//PRZYPISANIE BŁĘDÓW STACJI DO TABLICY 
aStationsErrors[1]															:=GeneralAlarms;											
aStationsErrors[2]															:=FormTransporterDispencerError;					//E_ConveyorState			// Transporter wjazdowy pod dozowniki
aStationsErrors[3]															:=FormTransporterScrewerError;						//E_ConveyorState			// Transporter wyjazdowy spod dozowników
aStationsErrors[4]															:=DispencersDragLeftError;							//E_DragStationState		// Przeciąganie formatek pod dozownikami
aStationsErrors[5]															:=DispencersCatch1Error;							//E_CatchStationState		// Chwytak butelek dozownika nr.1
aStationsErrors[6]															:=DispencersCatch2Error;							//E_CatchStationState		// Chwytak butelek dozownika nr.2
aStationsErrors[7]															:=DispencersCatch3Error;							//E_CatchStationState		// Chwytak butelek dozownika nr.3
aStationsErrors[8]															:=DispencersCatch4Error;							//E_CatchStationState		// Chwytak butelek dozownika nr.4				
aStationsErrors[9]															:=Dispencer1Error;									//E_DispencerState			// Dozownik 1
aStationsErrors[10]															:=Dispencer2Error;									//E_DispencerState			// Dozownik 2
aStationsErrors[11]															:=Dispencer3Error;									//E_DispencerState			// Dozownik 3							
aStationsErrors[12]															:=Dispencer4Error;									//E_DispencerState			// Dozownik 4
aStationsErrors[13]															:=TankHeatingError;									//E_MassHeatingState		// Grzanie masy
aStationsErrors[14]															:=WeightLiftError;									//E_WeightLiftState			// Podnoszenie wideł i szalek
aStationsErrors[15]															:=Weight1Error;										//E_WeightState				// Waga 1
aStationsErrors[16]															:=Weight2Error;										//E_WeightState				// Waga 2
aStationsErrors[17]															:=Weight3Error;										//E_WeightState				// Waga 3
aStationsErrors[18]															:=Weight4Error;										//E_WeightState				// Waga 4
aStationsErrors[19]															:=Dispencer1CorrectionError;						//E_WeightCorrectionState	//Korketa wagi 
aStationsErrors[20]															:=Dispencer2CorrectionError;						//E_WeightCorrectionState	//Korketa wagi 
aStationsErrors[21]															:=Dispencer3CorrectionError;						//E_WeightCorrectionState	//Korketa wagi 
aStationsErrors[22]															:=Dispencer4CorrectionError;						//E_WeightCorrectionState	//Korketa wagi 
aStationsErrors[23]															:=CapPuttedCheckError;								//E_CheckerState			// Sprawdzenie nałożenia nasadki
aStationsErrors[24]															:=GripperScrewerCatch1Error;						//E_CatchStationState 		// Łapanie butelek pod zakręcarkami 1
aStationsErrors[25]															:=GripperScrewerCatch2Error;						//E_CatchStationState 		// Łapanie butelek pod zakręcarkami	2
aStationsErrors[26]															:=GripperScrewer1Error;								//E_GriperScrewer			// Zakręcarka szczękowa 1
aStationsErrors[27]															:=GripperScrewer2Error;											
aStationsErrors[28]															:=BottleDragError;									//E_DragStationState		// Przeciąganie butelek pod zakręcarkami
aStationsErrors[29]															:=CapCorrectCheckError;								// E_CheckerState			// Sprawdzenie poprawności zakręcenia	
aStationsErrors[30]															:=BottleTransferError;								//E_BottleTransferState		// Robot
aStationsErrors[31]															:=GateRobotError;									// 							// Szlaban pod roobtem
aStationsErrors[32]															:=BadBottleConveyorError;							//E_ConvoyerState			// Stan transportera odrzuconych
aStationsErrors[33]															:=LabelMachineError;								// 							// Stan etykieciarki
aStationsErrors[34]															:=TanksError;										// 							// Stan zbiorników
aStationsErrors[35]															:=ExitTurnTableError;								//							// Stan stołu oboortowego wujscia z etykieciakri
aStationsErrors[36]															:=FormTransporterBeforeScrewerError;				//							// Spowalniacz formatek
aStationsErrors[37]															:=CapFeederError;									// Podajnik nasadek
aStationsErrors[38]															:=Weight5Error;										//E_WeightState				// Waga 5 	(** dodane 07.04.2022**)
aStationsErrors[39]															:=Weight6Error;										//E_WeightState				// Waga 6 	(** dodane 07.04.2022**)
aStationsErrors[40]															:=BottleFeederError;								// E_BottleFeederState     (** dodane 13.04.2022**)
aStationsErrors[41]															:=DispencersDragRightError;							//							// Przeciąganie formatek pod dozownikami prawa storna
aStationsErrors[42]															:=BarrierBetweenDispencers;							// 							//	Szlaban pod dozownikami od dwufazy
aStationsErrors[43]															:=BarrierBetweenWeights;
aStationsErrors[44]															:=BottleFeederTurnTableError;						//							//	Szlaban pomiedzy wagami od dwufazy
aStationsErrors[45]															:=BottleFeederFormGateError;
aStationsErrors[46]															:=SensorAcetoneError;
aStationsErrors[47]															:=SensorAirFlowError;
aStationsErrors[48]															:=LidFeederFormPositioningError;

aStationsErrors[49].bReset;
aStationsErrors[49].bError													:= stBottleSorterRead.eError.bError;
aStationsErrors[49].nErrorCode												:= stBottleSorterRead.eError.nErrorCode;
aStationsErrors[49].sErrorString											:= stBottleSorterRead.eError.sErrorString;
aStationsErrors[49].sErrorString2											:= stBottleSorterRead.eError.sErrorString2;
aStationsErrors[49].udiStationID											:= stBottleSorterRead.eError.udiStationID;
aStationsErrors[49].sStationName											:= Concat('Sorter butelek | ',stBottleSorterRead.eError.sStationName);

aStationsErrors[50].bReset;
aStationsErrors[50].bError													:= stCapSorterRead.eError.bError;
aStationsErrors[50].nErrorCode												:= stCapSorterRead.eError.nErrorCode;
aStationsErrors[50].sErrorString											:= stCapSorterRead.eError.sErrorString;
aStationsErrors[50].sErrorString2											:= stCapSorterRead.eError.sErrorString2;
aStationsErrors[50].udiStationID											:= stCapSorterRead.eError.udiStationID;
aStationsErrors[50].sStationName											:= Concat('Sorter nasadek | ',stCapSorterRead.eError.sStationName);

aStationsErrors[51]															:=CapSorterDragError;									
aStationsErrors[52]															:=BottlePusherError;									

aStationsErrors[53]															:=BarrierLidFeeder;	
aStationsErrors[54]															:=LidFeederError;		
aStationsErrors[55]															:=LidFeeder2Error;		
aStationsErrors[56]															:=LidFeederDragError;
aStationsErrors[57]															:=CapCorrectCheckCameraError;
aStationsErrors[58]															:=LidSealerError;		
aStationsErrors[59]															:=LidSealer2Error;		
aStationsErrors[60]															:=LidSealerDragError;

aStationsErrors[61]															:=PucksInserterError;		
aStationsErrors[62]															:=//PucksInserterTurnTableError;
aStationsErrors[63]															:=PucksInserterFormGateError;

aStationsErrors[64]															:=ROPPSlowerError;	
aStationsErrors[65]															:=ROPPFeederError;	
aStationsErrors[66]															:=ROPPDragError;	
aStationsErrors[67]															:=ROPPCappingError;
aStationsErrors[68]															:=FormTransporterROPPError;
aStationsErrors[69]															:=FormTransporterSlowerError;
aStationsErrors[70]															:=ExitConveyorError;
aStationsErrors[71]															:=SensorAcetoneError;
aStationsErrors[72]															:=SensorAirFlowError;
aStationsErrors[73]															:=ExhaustFanError;
aStationsErrors[79]															:= PucksInserterPushTableError_m1;
aStationsErrors[80]															:= PucksInserterPushTableError_m2;
aStationsErrors[81]															:= PucksInserterPushTableError_m3;
aStationsErrors[82];
aStationsErrors[83]															:= FormTransporterAfterScrewerError;
//Przegląd czy jakaś stacja jest w stanie błędu
aStationsErrors[84]															:= BottleTransferAfterDragError;
aStationsErrors[85] 														:= WickFeederError;
aStationsErrors[86]															:= WickFeederDragError;
aStationsErrors[87]															:= FormTransporterAfterCapSorterError;
aStationsErrors[88]															:= FormTransporterAfterBottleTransferError;
FOR i:=1 TO STATION_COUNT DO
	//Jeśli w stanie błędu
	
	IF aStationsErrors[i].bError THEN
		
		tonResetOff(IN:=bResetError,PT:=T#2S);
		
		IF tonResetOff.Q THEN
			aStationsErrors[i].bReset										:=FALSE;
			bResetError														:=FALSE;
		END_IF
		
		IF VIS.bResetErrorVisuCmd THEN
			aStationsErrors[i].bReset										:=TRUE;
			VIS.bResetErrorVisuCmd											:=FALSE;
		END_IF
		
		VIS.bErrorOccure													:=aStationsErrors[i].bError;
		bResetError															:=aStationsErrors[i].bReset;
		VIS.udiStationInError												:=aStationsErrors[i].udiStationID;
		VIS.sStationInError													:=aStationsErrors[i].sStationName;
		VIS.udiStationErrorCode												:=aStationsErrors[i].nErrorCode;
		VIS.sStationErrorDescription										:=aStationsErrors[i].sErrorString;
		VIS.sStationErrorDescription2										:=aStationsErrors[i].sErrorString2;
		EXIT;
		
	ELSE
		tonResetOff(IN:=bResetError,PT:=T#2S);
		//Jesli nie
		aStationsErrors[i].bError											:=FALSE;
		aStationsErrors[i].bReset											:=FALSE;
		aStationsErrors[i].sStationName										:='';
		aStationsErrors[i].nErrorCode										:=0;
		aStationsErrors[i].sErrorString										:='';
		aStationsErrors[i].sErrorString2									:='';
		VIS.bErrorOccure													:=FALSE;
	END_IF
	
	IF i>=60 THEN
		bResetError															:=FALSE;
	END_IF
	
END_FOR

// Zachowanie linii po wystapieniu błędu
IF VIS.bErrorOccure THEN
    VIS.bCycleStart 														:= FALSE; //DO WIZARDA
ELSE
    VIS.bErrorOccure              											:= FALSE;
    bResetError                  											:= FALSE;
    VIS.sStationInError           											:= '';
	VIS.udiStationInError													:=	0;
    VIS.udiStationErrorCode         										:= 0;
    VIS.sStationErrorDescription  											:= '';
    VIS.sStationErrorDescription2 											:= '';
    VIS.bResetErrorVisuCmd        											:= FALSE;
END_IF

// 
GeneralAlarms						:=aStationsErrors[1];										
FormTransporterDispencerError		:=aStationsErrors[2];					//E_ConveyorState			// Transporter wjazdowy pod dozowniki
FormTransporterScrewerError			:=aStationsErrors[3];					//E_ConveyorState			// Transporter wyjazdowy spod dozowników
DispencersDragLeftError				:=aStationsErrors[4];					//E_DragStationState		// Przeciąganie formatek pod dozownikami
DispencersCatch1Error				:=aStationsErrors[5];					//E_CatchStationState		// Chwytak butelek dozownika nr.1
DispencersCatch2Error				:=aStationsErrors[6];					//E_CatchStationState		// Chwytak butelek dozownika nr.2
DispencersCatch3Error				:=aStationsErrors[7];					//E_CatchStationState		// Chwytak butelek dozownika nr.3
DispencersCatch4Error				:=aStationsErrors[8];					//E_CatchStationState		// Chwytak butelek dozownika nr.4				
Dispencer1Error						:=aStationsErrors[9];					//E_DispencerState			// Dozownik 1
Dispencer2Error						:=aStationsErrors[10];					//E_DispencerState			// Dozownik 2
Dispencer3Error						:=aStationsErrors[11];					//E_DispencerState			// Dozownik 3							
Dispencer4Error						:=aStationsErrors[12];					//E_DispencerState			// Dozownik 4
TankHeatingError					:=aStationsErrors[13];					//E_MassHeatingState		// Grzanie masy
WeightLiftError						:=aStationsErrors[14];					//E_WeightLiftState			// Podnoszenie wideł i szalek
Weight1Error						:=aStationsErrors[15];					//E_WeightState				// Waga 1
Weight2Error						:=aStationsErrors[16];					//E_WeightState				// Waga 2
Weight3Error						:=aStationsErrors[17];					//E_WeightState				// Waga 3
Weight4Error						:=aStationsErrors[18];					//E_WeightState				// Waga 4
Dispencer1CorrectionError			:=aStationsErrors[19];				
Dispencer2CorrectionError			:=aStationsErrors[20];	
Dispencer3CorrectionError			:=aStationsErrors[21];	
Dispencer4CorrectionError			:=aStationsErrors[22];		
CapPuttedCheckError					:=aStationsErrors[23];					//E_CheckerState			// Sprawdzenie nałożenia nasadki
GripperScrewerCatch1Error			:=aStationsErrors[24];					//E_CatchStationState 		// Łapanie butelek pod zakręcarkami 1
GripperScrewerCatch2Error			:=aStationsErrors[25];					//E_CatchStationState 		// Łapanie butelek pod zakręcarkami	2
GripperScrewer1Error				:=aStationsErrors[26];					//E_GriperScrewer			// Zakręcarka szczękowa 1
GripperScrewer2Error			  	:=aStationsErrors[27];					//E_GriperScrewer			// Byyła Zakręcarka szczękowa 2;							
BottleDragError						:=aStationsErrors[28];					//E_DragStationState		// Przeciąganie butelek pod zakręcarkami
CapCorrectCheckError				:=aStationsErrors[29];					//E_CheckerState			// Sprawdzenie poprawności zakręcenia	
BottleTransferError					:=aStationsErrors[30];					// Robot
GateRobotError						:=aStationsErrors[31];			
BadBottleConveyorError				:=aStationsErrors[32];			
LabelMachineError					:=aStationsErrors[33];	
TanksError							:=aStationsErrors[34];	
ExitTurnTableError					:=aStationsErrors[35];	
FormTransporterBeforeScrewerError	:=aStationsErrors[36];	
CapFeederError						:=aStationsErrors[37];					// Podajnik nakrętek
Weight5Error						:=aStationsErrors[38];  				(** dodane 07.04.2022**)
Weight6Error						:=aStationsErrors[39];					(** dodane 07.04.2022**)
BottleFeederError					:=aStationsErrors[40];					(** dodane 13.04.2022**)
DispencersDragRightError			:=aStationsErrors[41];	
BarrierBetweenDispencers			:=aStationsErrors[42];
BarrierBetweenWeights				:=aStationsErrors[43];
BottleFeederTurnTableError			:=aStationsErrors[44];
BottleFeederFormGateError				:=aStationsErrors[45];
SensorAcetoneError 					:=aStationsErrors[46];
SensorAirFlowError 					:=aStationsErrors[47];
LidFeederFormPositioningError		:=aStationsErrors[48];	
stBottleSorterWrite.eError.bReset   :=aStationsErrors[49].bReset;						
stCapSorterWrite.eError.bReset   	:=aStationsErrors[50].bReset;	
CapSorterDragError					:=aStationsErrors[51];		
BottlePusherError					:=aStationsErrors[52];		
BarrierLidFeeder					:=aStationsErrors[53];												
LidFeederError						:=aStationsErrors[54];												
LidFeeder2Error						:=aStationsErrors[55];												
LidFeederDragError					:=aStationsErrors[56];											
CapCorrectCheckCameraError			:=aStationsErrors[57];											
LidSealerError						:=aStationsErrors[58];												
LidSealer2Error						:=aStationsErrors[59];												
LidSealerDragError					:=aStationsErrors[60];											

PucksInserterError					:=aStationsErrors[61];
//PucksInserterTurnTableError			:=aStationsErrors[62];
PucksInserterFormGateError			:=aStationsErrors[63];
ROPPSlowerError 					:=aStationsErrors[64];			
ROPPFeederError 					:=aStationsErrors[65];
ROPPDragError 						:=aStationsErrors[66];
ROPPCappingError 					:=aStationsErrors[67];
FormTransporterROPPError			:=aStationsErrors[68];
FormTransporterSlowerError			:=aStationsErrors[69];
ExitConveyorError					:=aStationsErrors[70];
SensorAcetoneError					:=aStationsErrors[71];
SensorAirFlowError					:=aStationsErrors[72];
ExhaustFanError						:=aStationsErrors[73];
PucksInserterPushTableError_m1		:=aStationsErrors[79];								
PucksInserterPushTableError_m2		:=aStationsErrors[80];								
PucksInserterPushTableError_m3		:=aStationsErrors[81];
									aStationsErrors[82];
FormTransporterAfterScrewerError	:=aStationsErrors[83];
BottleTransferAfterDragError		:=aStationsErrors[84];
WickFeederError						:=aStationsErrors[85];
WickFeederDragError					:=aStationsErrors[86];
FormTransporterAfterCapSorterError	:= aStationsErrors[87];	
FormTransporterAfterBottleTransferError := aStationsErrors[88];
//Przepisywanie ostatnich błędów
IF rtMachineStateAborting.Q THEN
    nCountSaveLastError := nCountSaveLastError + 1;
    aLastStationsErrors := aStationsErrors;
END_IF
IF P00_PackML.fbPMLAuto.ePMLState = Tc3_PackML.E_PMLState.ePMLState_EXECUTE THEN
	aLastStationsErrors := aStationsErrors;
END_IF
aStationsErrors[30].breset;

ACTION aActiveWarnings:
//	AwsActiveWarningDescription								:ARRAY [0..63] OF STRING;	//  Aktywne ostrzeżenia
//	iActiveWarning											:INT;	// Ilość aktywnych ostrzeżeń		


AbActiveWarningDescription[0]	:=	VIS.uliWarningOccure.0;
AbActiveWarningDescription[1]	:=	VIS.uliWarningOccure.1;
AbActiveWarningDescription[2]	:=	VIS.uliWarningOccure.2;
AbActiveWarningDescription[3]	:=	VIS.uliWarningOccure.3;
AbActiveWarningDescription[4]	:=	VIS.uliWarningOccure.4;
AbActiveWarningDescription[5]	:=	VIS.uliWarningOccure.5;
AbActiveWarningDescription[6]	:=	VIS.uliWarningOccure.6;
AbActiveWarningDescription[7]	:=	VIS.uliWarningOccure.7;
AbActiveWarningDescription[8]	:=	VIS.uliWarningOccure.8;
AbActiveWarningDescription[9]	:=	VIS.uliWarningOccure.9;
AbActiveWarningDescription[10]	:=	VIS.uliWarningOccure.10;
AbActiveWarningDescription[11]	:=	VIS.uliWarningOccure.11;
AbActiveWarningDescription[12]	:=	VIS.uliWarningOccure.12;
AbActiveWarningDescription[13]	:=	VIS.uliWarningOccure.13;
AbActiveWarningDescription[14]	:=	VIS.uliWarningOccure.14;
AbActiveWarningDescription[15]	:=	VIS.uliWarningOccure.15;
AbActiveWarningDescription[16]	:=	VIS.uliWarningOccure.16;
AbActiveWarningDescription[17]	:=	VIS.uliWarningOccure.17;
AbActiveWarningDescription[18]	:=	VIS.uliWarningOccure.18;
AbActiveWarningDescription[19]	:=	VIS.uliWarningOccure.19;
AbActiveWarningDescription[20]	:=	VIS.uliWarningOccure.20;
AbActiveWarningDescription[21]	:=	VIS.uliWarningOccure.21;
AbActiveWarningDescription[22]	:=	VIS.uliWarningOccure.22;
AbActiveWarningDescription[23]	:=	VIS.uliWarningOccure.23;
AbActiveWarningDescription[24]	:=	VIS.uliWarningOccure.24;
AbActiveWarningDescription[25]	:=	VIS.uliWarningOccure.25;
AbActiveWarningDescription[26]	:=	VIS.uliWarningOccure.26;
AbActiveWarningDescription[41]	:=	VIS.uliWarningOccure.41;
AbActiveWarningDescription[42]	:=	VIS.uliWarningOccure.42;

AbActiveWarningDescription[27]	:=	VIS.uliWarningOccure.27;
AbActiveWarningDescription[28]	:=	VIS.uliWarningOccure.28;
AbActiveWarningDescription[29]	:=	VIS.uliWarningOccure.29;
AbActiveWarningDescription[30]	:=	VIS.uliWarningOccure.30;
AbActiveWarningDescription[31]	:=	VIS.uliWarningOccure.31;
AbActiveWarningDescription[32]	:=	VIS.uliWarningOccure.32;
AbActiveWarningDescription[33]	:=	VIS.uliWarningOccure.33;
AbActiveWarningDescription[34]	:=	VIS.uliWarningOccure.34;
AbActiveWarningDescription[35]	:=	VIS.uliWarningOccure.35;
AbActiveWarningDescription[36]	:=	VIS.uliWarningOccure.36;
AbActiveWarningDescription[37]	:=	VIS.uliWarningOccure.37;
AbActiveWarningDescription[38]	:=	VIS.uliWarningOccure.38;
AbActiveWarningDescription[39]	:=	VIS.uliWarningOccure.39;
AbActiveWarningDescription[40]	:=	VIS.uliWarningOccure.40;

tonActiveWarning	(IN:=NOT tonActiveWarning.Q, PT:=T#1S);

IF tonActiveWarning.Q THEN
	FOR i:=0 TO 63 DO	
		VIS.AwsActiveWarningDescription[i] 	:= "";
		VIS.AudiActiveWarningDescriptionID[i]	:= 0;
	END_FOR
	VIS.iActiveWarning	:=	0;
	
	FOR i:=0 TO 63 DO		 
		
		 IF  AbActiveWarningDescription[i] = 1 THEN		
 
			FOR j:=0 TO 63 DO 
				IF  VIS.AwsActiveWarningDescription[j] = "" THEN
					VIS.AwsActiveWarningDescription[j]		:=	F_StringToWstringPL(VIS.AsWarningDescription[i]);
					VIS.AudiActiveWarningDescriptionID[j]	:=	AudiActiveWarningDescriptionIDtemp[i];
					EXIT;
				END_IF
			END_FOR	
			
			VIS.iActiveWarning	:=	VIS.iActiveWarning	+	1;	
		 END_IF
	END_FOR
END_IF
END_ACTION

ACTION aAlarms:
VIS.fbAlarms(
	bEnable:= , 
	nLangId:= , 
	tcEventFilterBase:= , 
	arrActiveEvents=> , 
	arrLoggedEvents=> , 
	nActiveEvents=> , 
	nLoggedEvents=> , 
	bBusy=> );

//Aktywne
VIS.bErrorOccure;
VIS.fbAlarms.arrActiveEvents[1].stEventEntry.nEventId;VIS.fbAlarms.arrActiveEvents[1].wsEventText;
VIS.fbAlarms.arrActiveEvents[2].stEventEntry.nEventId;VIS.fbAlarms.arrActiveEvents[2].wsEventText;
VIS.fbAlarms.arrActiveEvents[3].stEventEntry.nEventId;VIS.fbAlarms.arrActiveEvents[3].wsEventText;
VIS.fbAlarms.arrActiveEvents[4].stEventEntry.nEventId;VIS.fbAlarms.arrActiveEvents[4].wsEventText;
VIS.fbAlarms.arrActiveEvents[5].stEventEntry.nEventId;VIS.fbAlarms.arrActiveEvents[5].wsEventText;
VIS.fbAlarms.arrActiveEvents[6].stEventEntry.nEventId;VIS.fbAlarms.arrActiveEvents[6].wsEventText;
VIS.fbAlarms.arrActiveEvents[7].stEventEntry.nEventId;VIS.fbAlarms.arrActiveEvents[7].wsEventText;

//Historyczne
VIS.fbAlarms.arrLoggedEvents[1].nTimeRaised;VIS.fbAlarms.arrLoggedEvents[1].stEventEntry.nEventId;VIS.fbAlarms.arrLoggedEvents[1].wsEventText;
VIS.fbAlarms.arrLoggedEvents[2].nTimeRaised;VIS.fbAlarms.arrLoggedEvents[2].stEventEntry.nEventId;VIS.fbAlarms.arrLoggedEvents[2].wsEventText;
VIS.fbAlarms.arrLoggedEvents[3].nTimeRaised;VIS.fbAlarms.arrLoggedEvents[3].stEventEntry.nEventId;VIS.fbAlarms.arrLoggedEvents[3].wsEventText;
VIS.fbAlarms.arrLoggedEvents[4].nTimeRaised;VIS.fbAlarms.arrLoggedEvents[4].stEventEntry.nEventId;VIS.fbAlarms.arrLoggedEvents[4].wsEventText;
VIS.fbAlarms.arrLoggedEvents[5].nTimeRaised;VIS.fbAlarms.arrLoggedEvents[5].stEventEntry.nEventId;VIS.fbAlarms.arrLoggedEvents[5].wsEventText;
VIS.fbAlarms.arrLoggedEvents[6].nTimeRaised;VIS.fbAlarms.arrLoggedEvents[6].stEventEntry.nEventId;VIS.fbAlarms.arrLoggedEvents[6].wsEventText;
VIS.fbAlarms.arrLoggedEvents[7].nTimeRaised;VIS.fbAlarms.arrLoggedEvents[7].stEventEntry.nEventId;VIS.fbAlarms.arrLoggedEvents[7].wsEventText;
END_ACTION

ACTION aCommunicationError:


iBottleSorterReadLastWatchdog	:=	stBottleSorterRead.iWatchdog;
	
iCapSorterReadLastWatchdog		:=	stCapSorterRead.iWatchdog;
END_ACTION

ACTION aGeneralAlarms:
// Alarm_0001	1	Error	Stop Awaryjny, sprawdź bezpieczeństwo, zresetuj przyciskiem na panelu			aGeneralAlarms
// Alarm_0002	2	Error	Bład systemu | Diagnostyka systemu wykryła błąd - uruchom ponownie			aGeneralAlarms
// Alarm_0003	3	Error	Błąd systemu | Sprawdź sterownik i połączenia sieciowe a następnie uruchom ponownie maszynę			aGeneralAlarms
// Alarm_0004	4	Error	Błąd uruchamiania stacji | Brak możliwość wyłączenia stacji - zresetuj zasilanie			aGeneralAlarms
// Alarm_0005	5	Error	Błąd bazowania | Zbyt długie bazowanie stacji - sprawdź urządzenia			aGeneralAlarms
// Alarm_0006	6	Error	Błąd zatrzymywania | Zbyt długie zatrzymywanie cyklu w trybie normalnym			aGeneralAlarms
// Alarm_0007	7	Error	Błąd zasilania | Zanik fazy, lub zła kolejność faz - sprawdź podłączenie {0}			aGeneralAlarms
// Alarm_0008	8	Error	Błąd zasilania DC | Alarm zasilacza 10G1 - sprawdź zasilanie			aGeneralAlarms
// Alarm_0009	9	Error	Błąd zasilania DC | Alarm zasilacza 10G2 - sprawdź zasilanie			aGeneralAlarms
// Alarm_0010	10	Error	Błąd sprężonego powietrza | Zbyt niskie ciśnienie zasilania sprężonego powietrza - zwiększ ciśnienie {0}			aGeneralAlarms
// Alarm_0011	11	Error	Błąd bezpieczników 24VDC | Jeden z bezpieczników w bloku FB1 uległ przepaleniu - wymień bezpiecznik			aGeneralAlarms
// Alarm_0012	12	Error	Błąd bezpieczników 24VDC | Jeden z bezpieczników w bloku FB2 uległ przepaleniu - wymień bezpiecznik			aGeneralAlarms
// Alarm_0013	13	Error	Błąd bezpieczników 24VDC | Jeden z bezpieczników w bloku FB3 uległ przepaleniu - wymień bezpiecznik			aGeneralAlarms
// Alarm_0014	14	Error	Serwowzmacniacz | Wyłączone zabezpieczenie silnikowe - sprawdż zabezpieczenie			aGeneralAlarms
// Alarm_0015	15	Error	Napęd transportera | Wyłączone zabezpieczenie silnikowe - sprawdż zabezpieczenie			aGeneralAlarms
// Alarm_0016	16	Error	Napęd obrotu stacji znakowania | Wyłączone zabezpieczenie silnikowe - sprawdż zabezpieczenie			aGeneralAlarms
// Alarm_0017	17	Error	Stacja wyjściowa | Niewyjęta butelka z formatki - usuń butelkę			aGeneralAlarms
// Alarm_0018	18	Error	Stacja wejściowa | Źle włozona butelka - popraw			aGeneralAlarms
// Alarm_0019	19	Error	Sterownik główny | Brak napięcia zasilania na module ST2 w szafie głównej - sprawdź bezpiecznik			aGeneralAlarms
// Alarm_0020	20	Error	Sterownik w szafie robota | Brak napięcia zasilania na module ST1 w szafie robota - sprawdź bezpiecznik			aGeneralAlarms
// Alarm_0021	21	Error	Sterownik w szafie robota | Brak napięcia E-Bus na module ST1 w szafie robota - sprawdź bezpiecznik			aGeneralAlarms
// Alarm_0022	22	Error	Stacja zakręcarek | Zablokowana formatka za zakręcarką sprawdź położenie			aGeneralAlarms
// Alarm_0023	23	Error	Napęd transportera | Wyłączone zabezpieczenie silnikowe - sprawdż zabezpieczenie			aGeneralAlarms
// Alarm_0024	24	Error	Napęd transportera | Wyłączone zabezpieczenie silnikowe - sprawdż zabezpieczenie			aGeneralAlarms
// Alarm_0025	25	Error	Napęd transportera | Wyłączone zabezpieczenie silnikowe - sprawdż zabezpieczenie 			aGeneralAlarms
// Alarm_0026	26	Error	Napęd transportera | Wyłączone zabezpieczenie silnikowe - sprawdż zabezpieczenie			aGeneralAlarms
// Alarm_0027	27	Error	Napęd stołu obrotowego | Wyłączone zabezpieczenie silnikowe - sprawdż zabezpieczenie			aGeneralAlarms
// Alarm_0028	28	Error	Transporter odrzuconych | Zapełniony transporter odrzuconych butelek			aGeneralAlarms
// Alarm_0029	29	Error	Stacja dozowników | Zablokowana formatka przy dozownikach od strony drzwi. Usuń formatki i opakowania			aGeneralAlarms
// Alarm_0030	30	Error	Stacja zakręcarek | Zablokowana lub źle ustawiona formatka przed zakręcarkami. Sprawdź ustawienie formatek oraz czujniki obecności			aGeneralAlarms
// Alarm_0031	31	Error	Stacja zakręcarek | Źle ustawione formatki przed zakręcarką. Sprawdź czujniki obecności formatek			aGeneralAlarms
// Alarm_0032	32	Error	Stacja dozowników |Źle ustawione formatki przy dozownikach od strony drzwi. Przesuń formatki za wagi			aGeneralAlarms
// Alarm_0033	33	Error	Podajnik zamknięć | Brak zamknięć w 8 butelkach - sprawdź sorter			aGeneralAlarms
// Alarm_0034	34	Error	Brak gotowości stacji | Zbyt długie przygotowywanie stacji do gotowości {0}			aGeneralAlarms
// Alarm_0035	35	Error	Stacja zakręcarek | Formatki nie są dosunięte do pozycji przeciągania - odblokuj (wypadła nakrętka)			aGeneralAlarms
// Alarm_0036	36	Error	Sorter butelek | Brak komunikacji ze sterownikiem - włącz zasilanie/sprawdź podłączenie			aGeneralAlarms
// Alarm_0037	37	Error	Sorter nasadek | Brak komunikacji ze sterownikiem - włącz zasilanie/sprawdź podłączenie			aGeneralAlarms
// Alarm_0038	38	Error	Sorter nasadek - przeciąganie | Formatki nie są dosunięte do pozycji przeciągania - odblokuj (wypadła nakrętka)			aGeneralAlarms
// Alarm_0039	39	Error	Układ bezpieczeństwa | Brak komunikacji z sorterem nasadek - włącz linie/sprawdź komunikacje			aGeneralAlarms
// Alarm_0040	40	Error	Układ bezpieczeństwa | Brak komunikacji z sorterem butelek - włącz linie/sprawdź komunikacje			aGeneralAlarms
// Alarm_0041	41	Error	Stacja dozowników | Formatki nie są dosunięte do pozycji przeciągania - odblokuj (wypadła butelka)			aGeneralAlarms
// Alarm_0042	42	Error	Napęd stołu odbiorczego | Wyłączone zabezpieczenie silnikowe - sprawdż zabezpieczenie			aGeneralAlarms
// Alarm_0043	43	Error	Stacja przeciągania dozowniki lewe | Pozycja podnośnika dozowników jest poniżej ustawionej			aGeneralAlarms
// Alarm_0044	44	Error	Stacja przeciągania dozowniki prawe | Pozycja podnośnika dozowników jest poniżej ustawionej			aGeneralAlarms
// Alarm_0045	45	Error	Brak kapsla/lub kilku pod rząd przed stacją ROPP , nałóż kapsle na butelki			General
// Alarm_0046	46	Error	Stacja ROPP | Zablokowana formatka za ROPP			General
// Alarm_0047	47	Error	Stacja zgrzewania platynek (opcja)| Zablokowana formatka za stacją			General
// Alarm_0048	48	Error	Stacja sortera nakrętek | Zablokowana formatka za sorterem			General
// Alarm_0049	49	Error	Stacja przeciągania dozowniki lewe | Formatki nie przeciągnięte	General
// Alarm_0050	50	Error	Stacja przeciągania dozowniki prawe | Formatki nie przeciągnięte			General



IF bAlarmInit THEN
    bAlarmInit := FALSE; 
	fbSourceInfo.Clear();
	fbSourceInfo.sName:='UBL50-GeneralAlarms';
	fbSourceInfo.nId:=0;	
	// Alarm_0001	1	Error	Stop Awaryjny, sprawdź bezpieczeństwo, zresetuj przyciskiem na panelu			aGeneralAlarms
    arfbAlarm[1].CreateEx(stEventEntry := TC_EVENTS.AlarmClass.Alarm_0001, bWithConfirmation:= FALSE,  ipSourceInfo:= fbSourceInfo); 
	// Alarm_0002	2	Error	Bład systemu | Diagnostyka systemu wykryła błąd - uruchom ponownie			aGeneralAlarms
	arfbAlarm[2].CreateEx(stEventEntry := TC_EVENTS.AlarmClass.Alarm_0002, bWithConfirmation:= FALSE,  ipSourceInfo:= fbSourceInfo); 
	// Alarm_0003	3	Error	Błąd systemu | Sprawdź sterownik i połączenia sieciowe a następnie uruchom ponownie maszynę			aGeneralAlarms
	arfbAlarm[3].CreateEx(stEventEntry := TC_EVENTS.AlarmClass.Alarm_0003, bWithConfirmation:= FALSE,  ipSourceInfo:= fbSourceInfo); 
	// Alarm_0004	4	Error	Błąd uruchamiania stacji | Brak możliwość wyłączenia stacji - zresetuj zasilanie			aGeneralAlarms
	arfbAlarm[4].CreateEx(stEventEntry := TC_EVENTS.AlarmClass.Alarm_0004, bWithConfirmation:= FALSE,  ipSourceInfo:= fbSourceInfo); 
	// Alarm_0005	5	Error	Błąd bazowania | Zbyt długie bazowanie stacji - sprawdź urządzenia			aGeneralAlarms
	arfbAlarm[5].CreateEx(stEventEntry := TC_EVENTS.AlarmClass.Alarm_0005, bWithConfirmation:= FALSE,  ipSourceInfo:= fbSourceInfo); 
	// Alarm_0006	6	Error	Błąd zatrzymywania | Zbyt długie zatrzymywanie cyklu w trybie normalnym			aGeneralAlarms
	arfbAlarm[6].CreateEx(stEventEntry := TC_EVENTS.AlarmClass.Alarm_0006, bWithConfirmation:= FALSE,  ipSourceInfo:= fbSourceInfo); 
	// Alarm_0007	7	Error	Błąd zasilania | Zanik fazy, lub zła kolejność faz - sprawdź podłączenie			aGeneralAlarms
	arfbAlarm[7].CreateEx(stEventEntry := TC_EVENTS.AlarmClass.Alarm_0007, bWithConfirmation:= FALSE,  ipSourceInfo:= fbSourceInfo); 
	// Alarm_0008	8	Error	Błąd zasilania DC | Alarm zasilacza 10G1 - sprawdź zasilanie			aGeneralAlarms
	arfbAlarm[8].CreateEx(stEventEntry := TC_EVENTS.AlarmClass.Alarm_0008, bWithConfirmation:= FALSE,  ipSourceInfo:= fbSourceInfo); 
	// Alarm_0009	9	Error	Błąd zasilania DC | Alarm zasilacza 10G2 - sprawdź zasilanie			aGeneralAlarms
	arfbAlarm[9].CreateEx(stEventEntry := TC_EVENTS.AlarmClass.Alarm_0009, bWithConfirmation:= FALSE,  ipSourceInfo:= fbSourceInfo); 
	// Alarm_0010	10	Error	Błąd sprężonego powietrza | Zbyt niskie ciśnienie zasilania sprężonego powietrza - zwiększ ciśnienie			aGeneralAlarms
	arfbAlarm[10].CreateEx(stEventEntry := TC_EVENTS.AlarmClass.Alarm_0010, bWithConfirmation:= FALSE,  ipSourceInfo:= fbSourceInfo); 
	// Alarm_0011	11	Error	Błąd bezpieczników 24VDC | Jeden z bezpieczników w bloku FB1 uległ przepaleniu - wymień bezpiecznik			aGeneralAlarms
	arfbAlarm[11].CreateEx(stEventEntry := TC_EVENTS.AlarmClass.Alarm_0011, bWithConfirmation:= FALSE,  ipSourceInfo:= fbSourceInfo); 
	// Alarm_0012	12	Error	Błąd bezpieczników 24VDC | Jeden z bezpieczników w bloku FB2 uległ przepaleniu - wymień bezpiecznik			aGeneralAlarms
	arfbAlarm[12].CreateEx(stEventEntry := TC_EVENTS.AlarmClass.Alarm_0012, bWithConfirmation:= FALSE,  ipSourceInfo:= fbSourceInfo); 
	// Alarm_0013	13	Error	Błąd bezpieczników 24VDC | Jeden z bezpieczników w bloku FB3 uległ przepaleniu - wymień bezpiecznik			aGeneralAlarms
	arfbAlarm[13].CreateEx(stEventEntry := TC_EVENTS.AlarmClass.Alarm_0013, bWithConfirmation:= FALSE,  ipSourceInfo:= fbSourceInfo); 
	// Alarm_0014	14	Error	Serwowzmacniacz | Wyłączone zabezpieczenie silnikowe - sprawdż zabezpieczenie			aGeneralAlarms
	arfbAlarm[14].CreateEx(stEventEntry := TC_EVENTS.AlarmClass.Alarm_0014, bWithConfirmation:= FALSE,  ipSourceInfo:= fbSourceInfo); 
	// Alarm_0015	15	Error	Napęd transportera | Wyłączone zabezpieczenie silnikowe - sprawdż zabezpieczenie			aGeneralAlarms
	//arfbAlarm[15].CreateEx(stEventEntry := TC_EVENTS.AlarmClass.Alarm_0015, bWithConfirmation:= FALSE,  ipSourceInfo:= fbSourceInfo); 
	// Alarm_0016	16	Error	Napęd obrotu stacji znakowania | Wyłączone zabezpieczenie silnikowe - sprawdż zabezpieczenie			aGeneralAlarms
	arfbAlarm[16].CreateEx(stEventEntry := TC_EVENTS.AlarmClass.Alarm_0016, bWithConfirmation:= FALSE,  ipSourceInfo:= fbSourceInfo); 
	// Alarm_0017	17	Error	Stacja wyjściowa | Niewyjęta butelka z formatki - usuń butelkę			aGeneralAlarms
	arfbAlarm[17].CreateEx(stEventEntry := TC_EVENTS.AlarmClass.Alarm_0017, bWithConfirmation:= FALSE,  ipSourceInfo:= fbSourceInfo); 
	// Alarm_0018	18	Error	Stacja wejściowa | Źle włozona butelka - popraw			aGeneralAlarms
	arfbAlarm[18].CreateEx(stEventEntry := TC_EVENTS.AlarmClass.Alarm_0018, bWithConfirmation:= FALSE,  ipSourceInfo:= fbSourceInfo); 
	// Alarm_0019	19	Error	Sterownik główny | Brak napięcia zasilania na module ST2 w szafie głównej - sprawdź bezpiecznik			aGeneralAlarms
	arfbAlarm[19].CreateEx(stEventEntry := TC_EVENTS.AlarmClass.Alarm_0019, bWithConfirmation:= FALSE,  ipSourceInfo:= fbSourceInfo); 
	// Alarm_0020	20	Error	Sterownik w szafie robota | Brak napięcia zasilania na module ST1 w szafie robota - sprawdź bezpiecznik			aGeneralAlarms
	arfbAlarm[20].CreateEx(stEventEntry := TC_EVENTS.AlarmClass.Alarm_0020, bWithConfirmation:= FALSE,  ipSourceInfo:= fbSourceInfo); 
	// Alarm_0021	21	Error	Sterownik w szafie robota | Brak napięcia E-Bus na module ST1 w szafie robota - sprawdź bezpiecznik			aGeneralAlarms
	arfbAlarm[21].CreateEx(stEventEntry := TC_EVENTS.AlarmClass.Alarm_0021, bWithConfirmation:= FALSE,  ipSourceInfo:= fbSourceInfo); 
	// Alarm_0022	22	Error	Stacja zakręcarek | Zablokowana formatka za zakręcarką sprawdź położenie			aGeneralAlarms
	arfbAlarm[22].CreateEx(stEventEntry := TC_EVENTS.AlarmClass.Alarm_0022, bWithConfirmation:= FALSE,  ipSourceInfo:= fbSourceInfo); 
	// Alarm_0023	23	Error	Napęd transportera | Wyłączone zabezpieczenie silnikowe - sprawdż zabezpieczenie			aGeneralAlarms
	//arfbAlarm[23].CreateEx(stEventEntry := TC_EVENTS.AlarmClass.Alarm_0023, bWithConfirmation:= FALSE,  ipSourceInfo:= fbSourceInfo); 
	// Alarm_0024	24	Error	Napęd transportera | Wyłączone zabezpieczenie silnikowe - sprawdż zabezpieczenie			aGeneralAlarms
	//arfbAlarm[24].CreateEx(stEventEntry := TC_EVENTS.AlarmClass.Alarm_0024, bWithConfirmation:= FALSE,  ipSourceInfo:= fbSourceInfo); 
	// Alarm_0025	25	Error	Napęd transportera | Wyłączone zabezpieczenie silnikowe - sprawdż zabezpieczenie 			aGeneralAlarms
	//arfbAlarm[25].CreateEx(stEventEntry := TC_EVENTS.AlarmClass.Alarm_0025, bWithConfirmation:= FALSE,  ipSourceInfo:= fbSourceInfo); 
	// Alarm_0026	26	Error	Napęd transportera | Wyłączone zabezpieczenie silnikowe - sprawdż zabezpieczenie			aGeneralAlarms
	//arfbAlarm[26].CreateEx(stEventEntry := TC_EVENTS.AlarmClass.Alarm_0026, bWithConfirmation:= FALSE,  ipSourceInfo:= fbSourceInfo); 
	// Alarm_0027	27	Error	Napęd stołu obrotowego | Wyłączone zabezpieczenie silnikowe - sprawdż zabezpieczenie			aGeneralAlarms
	arfbAlarm[27].CreateEx(stEventEntry := TC_EVENTS.AlarmClass.Alarm_0027, bWithConfirmation:= FALSE,  ipSourceInfo:= fbSourceInfo); 
	// Alarm_0028	28	Error	Transporter odrzuconych | Zapełniony transporter odrzuconych butelek			aGeneralAlarms
	arfbAlarm[28].CreateEx(stEventEntry := TC_EVENTS.AlarmClass.Alarm_0028, bWithConfirmation:= FALSE,  ipSourceInfo:= fbSourceInfo); 
	// Alarm_0029	29	Error	Stacja dozowników | Zablokowana formatka przy dozownikach od strony drzwi. Usuń formatki i opakowania			aGeneralAlarms
	arfbAlarm[29].CreateEx(stEventEntry := TC_EVENTS.AlarmClass.Alarm_0029, bWithConfirmation:= FALSE,  ipSourceInfo:= fbSourceInfo); 
	// Alarm_0030	30	Error	Stacja zakręcarek | Zablokowana lub źle ustawiona formatka przed zakręcarkami. Sprawdź ustawienie formatek oraz czujniki obecności			aGeneralAlarms
	arfbAlarm[30].CreateEx(stEventEntry := TC_EVENTS.AlarmClass.Alarm_0030, bWithConfirmation:= FALSE,  ipSourceInfo:= fbSourceInfo); 
	// Alarm_0031	31	Error	Stacja zakręcarek | Źle ustawione formatki przed zakręcarką. Sprawdź czujniki obecności formatek			aGeneralAlarms
	arfbAlarm[31].CreateEx(stEventEntry := TC_EVENTS.AlarmClass.Alarm_0031, bWithConfirmation:= FALSE,  ipSourceInfo:= fbSourceInfo); 
	// Alarm_0032	32	Error	Stacja dozowników |Źle ustawione formatki przy dozownikach od strony drzwi. Przesuń formatki za wagi			aGeneralAlarms
	arfbAlarm[32].CreateEx(stEventEntry := TC_EVENTS.AlarmClass.Alarm_0032, bWithConfirmation:= FALSE,  ipSourceInfo:= fbSourceInfo); 
	// Alarm_0033	33	Error	Podajnik zamknięć | Brak zamknięć w 8 butelkach - sprawdź sorter			aGeneralAlarms
	arfbAlarm[33].CreateEx(stEventEntry := TC_EVENTS.AlarmClass.Alarm_0033, bWithConfirmation:= FALSE,  ipSourceInfo:= fbSourceInfo); 
	// Alarm_0034	34	Error	Brak gotowości stacji | Zbyt długie przygotowywanie stacji do gotowości			aGeneralAlarms
	arfbAlarm[34].CreateEx(stEventEntry := TC_EVENTS.AlarmClass.Alarm_0034, bWithConfirmation:= FALSE,  ipSourceInfo:= fbSourceInfo); 
	// Alarm_0035	35	Error	Stacja zakręcarek | Formatki nie są dosunięte do pozycji przeciągania - odblokuj (wypadła nakrętka)			aGeneralAlarms
	arfbAlarm[35].CreateEx(stEventEntry := TC_EVENTS.AlarmClass.Alarm_0035, bWithConfirmation:= FALSE,  ipSourceInfo:= fbSourceInfo); 
	// Alarm_0036	36	Error	Sorter butelek | Brak komunikacji ze sterownikiem - włącz zasilanie/sprawdź podłączenie			aGeneralAlarms
	arfbAlarm[36].CreateEx(stEventEntry := TC_EVENTS.AlarmClass.Alarm_0036, bWithConfirmation:= FALSE,  ipSourceInfo:= fbSourceInfo); 
	// Alarm_0037	37	Error	Sorter nasadek | Brak komunikacji ze sterownikiem - włącz zasilanie/sprawdź podłączenie			aGeneralAlarms
	arfbAlarm[37].CreateEx(stEventEntry := TC_EVENTS.AlarmClass.Alarm_0037, bWithConfirmation:= FALSE,  ipSourceInfo:= fbSourceInfo); 
	// Alarm_0038	38	Error	Sorter nasadek - przeciąganie | Formatki nie są dosunięte do pozycji przeciągania - odblokuj (wypadła nakrętka)			aGeneralAlarms
	arfbAlarm[38].CreateEx(stEventEntry := TC_EVENTS.AlarmClass.Alarm_0038, bWithConfirmation:= FALSE,  ipSourceInfo:= fbSourceInfo); 
	// Alarm_0039	39	Error	Układ bezpieczeństwa | Brak komunikacji z sorterem nasadek - włącz linie/sprawdź komunikacje			aGeneralAlarms
	arfbAlarm[39].CreateEx(stEventEntry := TC_EVENTS.AlarmClass.Alarm_0039, bWithConfirmation:= FALSE,  ipSourceInfo:= fbSourceInfo); 
	// Alarm_0040	40	Error	Układ bezpieczeństwa | Brak komunikacji z sorterem butelek - włącz linie/sprawdź komunikacje			aGeneralAlarms
	arfbAlarm[40].CreateEx(stEventEntry := TC_EVENTS.AlarmClass.Alarm_0040, bWithConfirmation:= FALSE,  ipSourceInfo:= fbSourceInfo); 
	// Alarm_0041	41	Error	Stacja dozowników | Formatki nie są dosunięte do pozycji przeciągania - odblokuj (wypadła butelka)			aGeneralAlarms
	arfbAlarm[41].CreateEx(stEventEntry := TC_EVENTS.AlarmClass.Alarm_0041, bWithConfirmation:= FALSE,  ipSourceInfo:= fbSourceInfo); 
	// Alarm_0042	42	Error	Napęd stołu odbiorczego | Wyłączone zabezpieczenie silnikowe - sprawdż zabezpieczenie			aGeneralAlarms
	arfbAlarm[42].CreateEx(stEventEntry := TC_EVENTS.AlarmClass.Alarm_0042, bWithConfirmation:= FALSE,  ipSourceInfo:= fbSourceInfo); 
	// Alarm_0043	43	Error	Stacja przeciągania dozowniki lewe | Pozycja podnośnika dozowników jest poniżej ustawionej			aGeneralAlarms
	arfbAlarm[43].CreateEx(stEventEntry := TC_EVENTS.AlarmClass.Alarm_0043, bWithConfirmation:= FALSE,  ipSourceInfo:= fbSourceInfo); 
	// Alarm_0044	44	Error	Stacja przeciągania dozowniki prawe | Pozycja podnośnika dozowników jest poniżej ustawionej			aGeneralAlarms
	arfbAlarm[44].CreateEx(stEventEntry := TC_EVENTS.AlarmClass.Alarm_0044, bWithConfirmation:= FALSE,  ipSourceInfo:= fbSourceInfo); 
	// Alarm_0045	45	Error	Brak kapsla/lub kilku pod rząd przed stacją ROPP , nałóż kapsle na butelki			General
	arfbAlarm[45].CreateEx(stEventEntry := TC_EVENTS.AlarmClass.Alarm_0045, bWithConfirmation:= FALSE,  ipSourceInfo:= fbSourceInfo); 
	// Alarm_0046	46	Error	Stacja ROPP | Zablokowana formatka za ROPP			General
	arfbAlarm[46].CreateEx(stEventEntry := TC_EVENTS.AlarmClass.Alarm_0046, bWithConfirmation:= FALSE,  ipSourceInfo:= fbSourceInfo); 
	// Alarm_0047	47	Error	Stacja zgrzewania platynek (opcja)| Zablokowana formatka za stacją			General
	arfbAlarm[47].CreateEx(stEventEntry := TC_EVENTS.AlarmClass.Alarm_0047, bWithConfirmation:= FALSE,  ipSourceInfo:= fbSourceInfo); 
	// Alarm_0048	48	Error	Stacja sortera nakrętek | Zablokowana formatka za sorterem			General
	arfbAlarm[48].CreateEx(stEventEntry := TC_EVENTS.AlarmClass.Alarm_0048, bWithConfirmation:= FALSE,  ipSourceInfo:= fbSourceInfo); 
	// Alarm_0049	49	Error	Stacja przeciągania dozowniki lewe | Formatki nie przeciągnięte	General
	arfbAlarm[49].CreateEx(stEventEntry := TC_EVENTS.AlarmClass.Alarm_0049, bWithConfirmation:= FALSE,  ipSourceInfo:= fbSourceInfo); 
	// Alarm_0050	50	Error	Stacja przeciągania dozowniki prawe | Formatki nie przeciągnięte	General
	arfbAlarm[50].CreateEx(stEventEntry := TC_EVENTS.AlarmClass.Alarm_0050, bWithConfirmation:= FALSE,  ipSourceInfo:= fbSourceInfo); 
	// Wolne do 80
END_IF






//Timery alarmów
tonDCSupply1OK(IN:=NOT IbDCSupply1OK, PT:=T#2S);
tonDCSupply2OK(IN:=NOT IbDCSupply2OK, PT:=T#2S);
tonDCSupply3OK(IN:=NOT IbDCSupply3OK, PT:=T#2S);
tonFuseFB1OK(IN:=NOT IbFuseFB1OK, PT:=T#2S);
tonFuseFB2OK(IN:=NOT IbFuseFB2OK AND IbEmergencyStop, PT:=T#2S);
tonEmergencyStop(IN:=IbEmergencyStop, PT:=T#4S);
tonFirstCycle(IN:=bFirstCycle, PT:=T#10S);	
tonSystemDiagnosisError(IN:=P00_SystemDiagnostics.bError AND tonFirstCycle.Q (*AND NOT GeneralAlarms.bError*), PT:=T#200S);																// zmniejszyłem czas do 20MS, bo przy 50MS butelka potrafiła przejechać. 
tonCompressedAir(IN:= (NOT IbCompressedAirOK OR NOT GVL_IO.IbPressureInSystemSensor) AND IbEmergencyStop(*OR NOT P07_ROPP.IbROPPCompressedAirOK*) (*AND NOT GeneralAlarms.bError*) AND NOT VIS.bCapCorrectCheckIgnoreErrors , PT:=T#5S);

tonBottleCheckAfterBottleTransferSensor	(IN:=P13_BottleTransfer.IbBottleCheckAfterBottleTransferSensor	AND P00_PackML.tofTransportersWorking.Q ,PT:=T#20MS); //Alarm niewyjętej butelki, wcześniej był zależy od włączonego robta
tonIbBottleNotInserted					(IN:=P01_BottleFeeder.IbBottleFeederNotInsertedSensor 						AND P00_PackML.tofTransportersWorking.Q ,PT:=T#20MS); 
tonPowerSuppyTerminal1UsUndervoltageError(IN:=IbPowerSuppyTerminal1UsUndervoltage, PT:=T#3S);
tonPowerSuppyTerminal2UpUndervoltageError(IN:=IbPowerSuppyTerminal2UpUndervoltage, PT:=T#3S);
tonPowerSuppyTerminal2UsUndervoltageError(IN:=IbPowerSuppyTerminal2UsUndervoltage, PT:=T#3S);

 //Watchdogi 
TimerWatchdog_eUndefined  					(IN :=		P00_PackML.fbPMLModeManager.eModeStatus = E_PMLUnitMode.ePMLUnitMode_UNDEFINED, 								PT:=T#30S);
TimerWatchdog_eAborting						(IN	:=		P00_PackML.fbPMLAuto.ePMLState = E_PMLState.ePMLState_ABORTING, 												PT:=T#30S);
TimerWatchdog_eResetting					(IN	:=		P00_PackML.fbPMLAuto.ePMLState = E_PMLState.ePMLState_RESETTING AND P00_PackML.bHomingIsOnAtLeastOneStation, 	PT:=T#2M);
TimerWatchdog_eStopping						(IN	:=		P00_PackML.fbPMLAuto.ePMLState = E_PMLState.ePMLState_STOPPING, 												PT:=T#15S);
TimerWatchdog_eIdleAndNotStationsAreReady	(IN	:=		P00_PackML.fbPMLAuto.ePMLState = E_PMLState.ePMLState_IDLE AND 
													NOT (P00_PackML.fbPMLModeManager.eModeStatus = E_PMLUnitMode.ePMLUnitMode_MANUAL) AND
													NOT	P00_PackML.bStationsAreReady
																																										,PT:=T#3S); 

//Czujnik zapełnienia odrzutów 28.05
tonBadBottleConvoyerAlarm(IN:=P14_BadBottleConyevor.IbBadBottleConveyorFullSensor, PT:=T#3M); // było 6
tonBadBottleConvoyerAlarm.ET;

//Alarm zablokowanej formatki przed dozownikiem
tonFormStuckBeforeDispencer14Alarm( IN:=
										(
										NOT bDosingTwoPhases AND
											(
												(	MAIN.IbFourthFormCheckFormSensor AND NOT MAIN.IbSecondFormCheckFormSensor) OR
												(P00_PackML.iGateDispCase = 600 AND VIS.bGateBeforeDispencersRun AND MAIN.IbFormCheckFormSensor)
											)
										)
										AND
										(P00_PackML.fbPMLAuto.ePMLState = E_PMLState.ePMLState_EXECUTE) AND P00_PackML.tonLongDelayAfterStart.Q , PT:=T#20S);

//Alarm zablokowanej formatki
tonFormStuckAfterDispencerAlarm(IN:=
									P00_PackML.tonLongDelayAfterStart.Q AND
									NOT bDosingTwoPhases AND
									(
										(
											(NOT P05_Weight.IbWeight1FormSensor OR NOT P05_Weight.IbWeight2FormSensor OR NOT P05_Weight.IbWeight3FormSensor OR NOT P05_Weight.IbWeight4FormSensor)  AND
											(eAfterDispencersPackageState[1].bFormPresent OR eAfterDispencersPackageState[2].bFormPresent OR 
											 eAfterDispencersPackageState[3].bFormPresent OR eAfterDispencersPackageState[4].bFormPresent OR P00_PackML.fbIbDispencerAfterCheckFormSensor.bOut) AND 
											 (P00_PackML.fbPMLAuto.ePMLState = E_PMLState.ePMLState_EXECUTE) AND
											 bFormTransportersScrewerCmdStart AND 
											 //bFormTransportersBeforeROPPCmdStart AND 
											NOT MAIN.IbLidSealerAfterSensor
										 ) 
									 	OR
									 (
											(NOT P05_Weight.IbWeight1FormSensor OR NOT P05_Weight.IbWeight2FormSensor OR NOT P05_Weight.IbWeight3FormSensor OR NOT P05_Weight.IbWeight4FormSensor)  AND
											MAIN.IbTwoPhasesFormSensorBetweenDispencers  AND 
											 (P00_PackML.fbPMLAuto.ePMLState = E_PMLState.ePMLState_EXECUTE) AND
											  bFormTransportersScrewerCmdStart AND 
											 //bFormTransportersBeforeROPPCmdStart AND 
											NOT MAIN.IbLidSealerAfterSensor
					 
									 )
									 )
									 {warning 'BLAD ZABL. FOR - ZMIANA DO SPRAWDZNENIA'}
									, PT:=T#20S);
																								 
//Alarm zablokowanej formatki za dozownikiam 34
tonFormStuckAfterDispencer34Alarm	(IN:=	(
												(
												NOT MAIN.IbTwoPhasesFormSensorBetweenDispencers AND (eBeforeDispencer12PackageState2Phase[1].bFormPresent OR eBeforeDispencer12PackageState2Phase[2].bFormPresent)
												) OR
												(
														 MAIN.IbTwoPhasesFormSensorBetweenDispencers AND 
													(
														(eAfterDispencer34PackageState2Phase[1].bFormPresent OR eAfterDispencer34PackageState2Phase[2].bFormPresent) AND
													 	eBeforeDispencer12PackageState2Phase[1].bFormPresent AND eBeforeDispencer12PackageState2Phase[2].bFormPresent
													)
												)
											) AND 
												((P00_PackML.fbPMLAuto.ePMLState = E_PMLState.ePMLState_EXECUTE) OR (P00_PackML.fbPMLAuto.ePMLState = E_PMLState.ePMLState_STOPPING))
										, PT:=T#60S); //? dp zwiekszony  czas

tonFormsStuckAfterLidSealerAlarm; 	{warning ' dorobic alarmy zablokowanych formatek'}
tonFormsStuckAfterROPPAlarm	;		{warning ' dorobic alarmy zablokowanych formatek'}
tonFormsStuckAfterCapSorterAlarm	(IN:= (P00_PackML.fbPMLAuto.ePMLState = E_PMLState.ePMLState_EXECUTE) AND bCapSorterDragEnable AND NOT P10_GripperScrewer.IbGripperScrewersThirdFormCheckFormSensor AND
											(MAIN.IbCapSorterAfterFormSensor OR MAIN.IbCapSorterAfterFormSensor2), PT:=T#10S);

//Alarm Zablokowanej formatki przed zakręcarkami
tonbFormsStuckBeforeScrewersAlarm( IN := P09_CapPuttedCheck.IbCapPuttedCheckFormSensor AND P10_GripperScrewer.IbGripperScrewersbeforeThirdFormCheckFormSensor AND //bylo bez before
										(NOT eBeforeScrewersPackageState[1].bFormPresent OR NOT eBeforeScrewersPackageState[2].bFormPresent OR
										 NOT eBeforeScrewers2PackageState[1].bFormPresent OR NOT eBeforeScrewers2PackageState[2].bFormPresent) AND
										(P00_PackML.fbPMLAuto.ePMLState = E_PMLState.ePMLState_EXECUTE) 
										, PT:=T#10S);
tonFormsStuckBeforeScrewersAlarm2( IN:= (NOT P10_GripperScrewer.IbGripperScrewersThirdFormCheckFormSensor AND eBeforeScrewersPackageState[1].bFormPresent AND eBeforeScrewersPackageState[2].bFormPresent AND
										 eBeforeScrewers2PackageState[1].bFormPresent AND  eBeforeScrewers2PackageState[2].bFormPresent) AND
										(P00_PackML.fbPMLAuto.ePMLState = E_PMLState.ePMLState_EXECUTE) AND P00_PackML.tonLongDelayAfterStart.Q , PT:=T#10S);
// Alarm nakretka wypadła pod zakrecarke	
tonFormsStuckBeforeScrewersAlarm3( IN:= P10_GripperScrewer.IbGripperScrewersBeforeThirdFormCheckFormSensor AND  
										//P00_PackML.fbIbGripperScrewersThirdFormCheckFormSensor.bOut AND//Gotowy do przeciągania
										(P00_PackML.fbPMLAuto.ePMLState = E_PMLState.ePMLState_EXECUTE) AND P00_PackML.tonLongDelayAfterStart.Q , PT:=T#10S);

// Zablokowana formatka za zakrecarka
iCounterFormsAfterScrewer:= BOOL_TO_INT(eAfterScrewerPackageState[1].bFormPresent)+
							BOOL_TO_INT(eAfterScrewerPackageState[2].bFormPresent);
//tonFormsStuckAfterScrewersAlarm(IN:=	(iCounterFormsAfterScrewer>=1 OR P11_CapCorrectCheck.IbCapCorrectCheckFormSensor OR (P11_CapCorrectCheck.IbCapCorrectCheckAfterScrewerFormSensor OR P11_CapCorrectCheck.IbCapCorrectCheckDialAfterScrewerFormSensor))
//														AND P00_PackML.fbPMLAuto.ePMLState = E_PMLState.ePMLState_EXECUTE
//														AND NOT P13_BottleTransfer.IbSecondFormCheckFormSensor
//								, PT:=T#10S);
tonFormsStuckAfterScrewersAlarm(IN:=	(P11_CapCorrectCheck.IbCapCorrectCheckAfterScrewerFormSensor OR P11_CapCorrectCheck.IbCapCorrectCheckDialAfterScrewerFormSensor) AND
										P00_PackML.fbPMLAuto.ePMLState = E_PMLState.ePMLState_EXECUTE AND
										NOT P13_BottleTransfer.IbSecondFormCheckFormSensor
								, PT:=T#20S);


						
tonFormsStuckBeforeCapSorterAlarm( IN:= (stCapSorterRead.eReservedSignals.bReserved00 OR
										(MAIN.IbCapSorterBeforeFourthFormCheckFormSensor AND NOT MAIN.IbCapSorterFirstFormCheckFormSensor) OR 
										(MAIN.IbCapSorterBeforeFourthFormCheckFormSensor  AND MAIN.IbCapSorterFirstFormCheckFormSensor AND NOT P00_PackML.fbIbCapSorterFourthFormCheckFormSensor.bOut) 
										
										)
										AND  
										//P00_PackML.fbIbGripperScrewersThirdFormCheckFormSensor.bOut AND//Gotowy do przeciągania
										(P00_PackML.fbPMLAuto.ePMLState = E_PMLState.ePMLState_EXECUTE) AND P00_PackML.tonLongDelayAfterStart.Q , PT:=T#10S);

	
tonstBottleSorterReadiWatchdog	( IN:=	iBottleSorterReadLastWatchdog	=	stBottleSorterRead.iWatchdog	AND NOT bBottleSorterDisable,PT:= T#10S);
tonstBottleSorterReadiWatchdog.ET;
tonstCapSorterReadiWatchdog		( IN:=	iCapSorterReadLastWatchdog		=	stCapSorterRead.iWatchdog		AND NOT bCapSorterDisable,PT:= T#10S);	
tonstCapSorterReadiWatchdog.ET;

tonbFormsDragingLeftRunCheck	(IN:=bFormsDragingLeftRunCheck AND NOT VIS.bFormsDragingLeftRun,	PT:=T#100MS);
tonbFormsDragingRightRunCheck	(IN:=bFormsDragingRightRunCheck AND NOT VIS.bFormsDragingRightRun,	PT:=T#100MS);
//=========================================================================================================================================================	


tonResetFuseBlock(IN:=QbResetFuseFB1 OR QbResetFuseFB2 OR QbResetFuseFB3,PT:=T#2S);

IF tonResetFuseBlock.Q THEN
	QbResetFuseFB1:=QbResetFuseFB2:=QbResetFuseFB3:=FALSE;
END_IF

rtEmergencyStop(CLK:=NOT IbEmergencyStop,Q=>);





IF GeneralAlarms.bReset THEN
	
	// Alarm_0002	2	Error	Bład systemu | Diagnostyka systemu wykryła błąd - uruchom ponownie			aGeneralAlarms
	// BLAD 31 - Diagnostyka
	IF arfbAlarm[2].bActive THEN
		P00_SystemDiagnostics.bReset:=TRUE;	
		GeneralAlarms.bError:=FALSE;
	END_IF
	
	//Alarm_0006	6	Error	Błąd zatrzymywania | Zbyt długie zatrzymywanie cyklu w trybie normalnym
	// BLAD 35 - WatchDog stanu eStoping
	IF arfbAlarm[6].bActive THEN
		P00_PackML.ACT_ResetCommands();
		GeneralAlarms.bError:=FALSE;
	END_IF
	
	//Alarm_0011	11	Error	Błąd bezpieczników 24VDC | Jeden z bezpieczników w bloku FB1 uległ przepaleniu - wymień bezpiecznik
	//BŁĄD 40 - przepalony bezpiecznik FB1
	IF arfbAlarm[11].bActive THEN
		GeneralAlarms.bError:=FALSE;
		QbResetFuseFB1 := TRUE; 
	END_IF

	//Alarm_0012	12	Error	Błąd bezpieczników 24VDC | Jeden z bezpieczników w bloku FB2 uległ przepaleniu - wymień bezpiecznik
	//BŁĄD 41 - przepalony bezpiecznik FB2	zrobic timer
	IF arfbAlarm[12].bActive THEN
		GeneralAlarms.bError:=FALSE;
		QbResetFuseFB2 := TRUE; 
		QbResetFuseFB3 := TRUE; 
	END_IF
	
	//Alarm_0022	22	Error	Stacja zakręcarek | Zablokowana formatka za zakręcarką sprawdź położenie
	//BŁĄD 51 -	Zablokowana formatka przy stacji zakręcarek
	IF arfbAlarm[22].bActive THEN
		GeneralAlarms.bError:=FALSE;
		eAfterScrewerPackageState[1].bFormPresent:=FALSE;
		eAfterScrewerPackageState[2].bFormPresent:=FALSE;
	END_IF
	
	//Alarm_0030	30	Error	Stacja zakręcarek | Zablokowana lub źle ustawiona formatka przed zakręcarkami. Sprawdź ustawienie formatek oraz czujniki obecności
	//Błąd 59 zablokowanej formatki przed zakręcarkmi
	IF arfbAlarm[30].bActive THEN
		GeneralAlarms.bError:=FALSE;
		eAfterDispencer34PackageState2Phase[1].bFormPresent:=FALSE;
		eAfterDispencer34PackageState2Phase[2].bFormPresent:=FALSE;
		eBeforeDispencer12PackageState2Phase[1].bFormPresent:=FALSE;
		eBeforeDispencer12PackageState2Phase[2].bFormPresent:=FALSE;
	END_IF

	//Alarm_0032	32	Error	Stacja dozowników |Źle ustawione formatki przy dozownikach od strony drzwi. Przesuń formatki za wagi
	//Błąd 61 zablokowanej formatki za dozownikami
	IF arfbAlarm[32].bActive THEN
		eAfterDispencersPackageState[1].bFormPresent	:=	FALSE;
		eAfterDispencersPackageState[2].bFormPresent	:=	FALSE;
		eAfterDispencersPackageState[3].bFormPresent	:=	FALSE;
		eAfterDispencersPackageState[4].bFormPresent	:=	FALSE;			
		GeneralAlarms.bError							:=	FALSE;
	END_IF
	
	//Alarm_0033	33	Error	Podajnik zamknięć | Brak zamknięć w 8 butelkach - sprawdź sorter
	//BŁĄD 62 - Brak nasadek po sorterze 
	//wykomentowany błąd 8 butelek	
	IF arfbAlarm[33].bActive THEN	
		GeneralAlarms.bError		:=	FALSE;
		iCapFeederCheckCountNOK		:=	0;
	END_IF

	//Alarm_0034	34	Error	Brak gotowości stacji | Zbyt długie przygotowywanie stacji do gotowości
	// BLAD 63 - WatchDog stanu Idle ale bez gotowych stacji
	IF arfbAlarm[34].bActive THEN
		P00_PackML.ACT_ResetCommands();
		GeneralAlarms.bError		:=FALSE;
	END_IF

	// Alarm_0049	49	Error	Stacja przeciągania dozowniki lewe | Formatki nie przeciągnięte	General
	// Alarm_0050	50	Error	Stacja przeciągania dozowniki prawe | Formatki nie przeciągnięte	General	
	IF arfbAlarm[49].bActive OR arfbAlarm[50].bActive THEN
        eBeforeDispencersPackageState[4].bDoseAborted:=TRUE;eDispencersPackageState[4].bDoseAborted:=TRUE;
        eBeforeDispencersPackageState[3].bDoseAborted:=TRUE;eDispencersPackageState[3].bDoseAborted:=TRUE;
        eBeforeDispencersPackageState[2].bDoseAborted:=TRUE;eDispencersPackageState[2].bDoseAborted:=TRUE;
        eBeforeDispencersPackageState[1].bDoseAborted:=TRUE;eDispencersPackageState[1].bDoseAborted:=TRUE;				
		eDispencer12PackageState2Phase[1].bDoseAbortedSecondPhase:=TRUE;	eDispencer12PackageState2Phase[1].bDoseAborted:=TRUE;		
		eDispencer12PackageState2Phase[2].bDoseAbortedSecondPhase:=TRUE;	eDispencer12PackageState2Phase[2].bDoseAborted:=TRUE;				
		eDispencer34PackageState2Phase[1].bDoseAborted:=TRUE;	eDispencer34PackageState2Phase[1].bDoseAbortedSecondPhase:=TRUE;	
		eDispencer34PackageState2Phase[2].bDoseAborted:=TRUE;	eDispencer34PackageState2Phase[2].bDoseAbortedSecondPhase:=TRUE;	
		P00_PackML.ACT_ResetCommands();
		GeneralAlarms.bError		:=FALSE;
	END_IF

	IF arfbAlarm[50].bActive THEN
		P00_PackML.ACT_ResetCommands();
		GeneralAlarms.bError		:=FALSE;
	END_IF
	
	GeneralAlarms.bError		:=FALSE;
	
	CASE GeneralAlarms.nErrorCode OF
		
// 		31: 	
// 			GeneralAlarms.bError:=FALSE;
// 			P00_SystemDiagnostics.bReset:=TRUE;			
			
// 		33:	// BLAD 4 - WatchDog stanu eAborting
// 			{warning 'Dorobić wyjście z eAborting'}
// 			GeneralAlarms.bError:=FALSE;

// 		35: // BŁAD 6 Zatrzymywania, kasowanie wszystkich rozkazów
// 			P00_PackML.ACT_ResetCommands();
// 			GeneralAlarms.bError:=FALSE;

// 		40: //Bezpieczniki 1
// 			GeneralAlarms.bError:=FALSE;
// 			QbResetFuseFB1 := TRUE; 
			
// 		41://Bezpieczniki 2
// 			GeneralAlarms.bError:=FALSE;
// 			QbResetFuseFB2 := TRUE; 
// 			QbResetFuseFB3 := TRUE; 
// 		42://Bezpieczniki 3
// 			GeneralAlarms.bError:=FALSE;		
// 		51:
// 			GeneralAlarms.bError:=FALSE;
// 			//nCountertooLong:=nCountertooLong+1;
// 			//IF nCountertooLong>=1 THEN
// 				eAfterScrewerPackageState[1].bFormPresent:=FALSE;
// 				eAfterScrewerPackageState[2].bFormPresent:=FALSE;
// 			//	nCountertooLong:=0;
// 			//END_IF
// 		59:
// 			GeneralAlarms.bError:=FALSE;
// 			eAfterDispencer34PackageState2Phase[1].bFormPresent:=FALSE;
// 			eAfterDispencer34PackageState2Phase[2].bFormPresent:=FALSE;
// 			eBeforeDispencer12PackageState2Phase[1].bFormPresent:=FALSE;
// 			eBeforeDispencer12PackageState2Phase[2].bFormPresent:=FALSE;
// 
// 		61: //Stacja dozowników|ŹLE ustawione formatki przy dozownikach od strony drzwi. Przesuń formatki za wagi
// 			eAfterDispencersPackageState[1].bFormPresent	:=	FALSE;
// 			eAfterDispencersPackageState[2].bFormPresent	:=	FALSE;
// 			eAfterDispencersPackageState[3].bFormPresent	:=	FALSE;
// 			eAfterDispencersPackageState[4].bFormPresent	:=	FALSE;			
// 			GeneralAlarms.bError							:=	FALSE;
	
// 		62: //Brak podawania nasadek		
// 			GeneralAlarms.bError		:=	FALSE;
// 			iCapFeederCheckCountNOK		:=	0;
// 			
// 		63: //Bład 36 Idle i Not Ready
// 			P00_PackML.ACT_ResetCommands();
// 			GeneralAlarms.bError		:=FALSE;
			
			
		368: //Blad brak nasadki ROPP
			GeneralAlarms.bError								:= FALSE;
			eBeforeROPPCapControlPackageState[1].bROPPPutted 	:= TRUE;
			eBeforeROPP2PackageState[3].bROPPPutted				:= TRUE;
			eBeforeROPP2PackageState[2].bROPPPutted				:= TRUE;
			eBeforeROPP2PackageState[1].bROPPPutted				:= TRUE;
			eBeforeROPPPackageState[2].bROPPPutted				:= TRUE;	
			eBeforeROPPPackageState[1].bROPPPutted				:= TRUE;			
			GVL_ROPP.iROPPFeederCheckCountNOK					:= 0;
		369: // Stacja ROPP | Zablokowana formatka za ROPP
			GeneralAlarms.bError		:=FALSE;
		370: // Stacja zgrzewania platynek (opcja)| Zablokowana formatka za stacją
			GeneralAlarms.bError		:=FALSE;
		371: // Stacja sortera nakrętek | Zablokowana formatka za sorterem
			GeneralAlarms.bError		:=FALSE;
		ELSE
			GeneralAlarms.bError		:=FALSE;
	END_CASE
	
END_IF

// Alarm_0001	1	Error	Stop Awaryjny, sprawdź bezpieczeństwo, zresetuj przyciskiem na panelu			aGeneralAlarms
//BŁĄD 1 - Stop Awaryjny
//IF NOT IbEmergencyStop THEN
IF NOT IbEmergencyStop AND NOT tonSystemDiagnosisError.Q AND NOT bBottleSorterSystemDiagError THEN
	IF NOT arfbAlarm[1].bActive THEN
		arfbAlarm[1].Raise(nTimeStamp:=0);
	END_IF
	
//	GVL_ErrorHandling.stGeneralAlarms.bReset:=FALSE;
//	GVL_Unit.eCommand := E_PackMLCommand.eAbort; 

	ELSE //opcja z autoresetem
	IF arfbAlarm[1].bActive THEN
		arfbAlarm[1].Clear(nTimeStamp:=0, bResetConfirmation:= FALSE);	
	END_IF	

		
END_IF	

// Alarm_0002	2	Error	Bład systemu | Diagnostyka systemu wykryła błąd - uruchom ponownie			aGeneralAlarms
// BLAD 31 - Diagnostyka
IF tonSystemDiagnosisError.Q THEN
	IF NOT arfbAlarm[2].bActive THEN
		arfbAlarm[2].Raise(nTimeStamp:=0);
	END_IF
	ELSE
	IF arfbAlarm[2].bActive AND GeneralAlarms.bReset THEN
		arfbAlarm[2].Clear(nTimeStamp:=0, bResetConfirmation:= FALSE);	
	END_IF	
// 	GeneralAlarms.bError:=TRUE;
// 	GeneralAlarms.bReset:=FALSE;
// 	GeneralAlarms.nErrorCode:=31;
// 	GeneralAlarms.udiStationID:=1;	
// 	GeneralAlarms.sStationName:='Błąd systemu';
// 	GeneralAlarms.sErrorString:='Bład systemu | Diagnostyka systemu wykryła błąd - uruchom ponownie';	
// 	GeneralAlarms.sErrorString2:=Concat(WSTRING_TO_STRING(P00_SystemDiagnostics.sErrorDescription),UDINT_TO_STRING(P00_SystemDiagnostics.udiErrorID));	
END_IF

//Alarm_0003	3	Error	Błąd systemu | Sprawdź sterownik i połączenia sieciowe a następnie uruchom ponownie maszynę
// BLAD 32 - WatchDog stanu Undefined
IF TimerWatchdog_eUndefined.Q THEN
	IF NOT arfbAlarm[3].bActive THEN
		arfbAlarm[3].Raise(nTimeStamp:=0);
	END_IF
	ELSE
	IF arfbAlarm[3].bActive AND GeneralAlarms.bReset THEN
		arfbAlarm[3].Clear(nTimeStamp:=0, bResetConfirmation:= FALSE);	
	END_IF
// 	GeneralAlarms.bError:=TRUE;
// 	GeneralAlarms.bReset:=FALSE;
// 	GeneralAlarms.nErrorCode:=32;
// 	GeneralAlarms.udiStationID:=1;		
// 	GeneralAlarms.sStationName:='Błąd systemu';
// 	GeneralAlarms.sErrorString:='Błąd systemu | Sprawdź sterownik i połączenia sieciowe a następnie uruchom ponownie maszynę';	
END_IF

//Alarm_0004	4	Error	Błąd uruchamiania stacji | Brak możliwość wyłączenia stacji - zresetuj zasilanie
// BLAD 33 - WatchDog stanu eAborting
IF TimerWatchdog_eAborting.Q THEN
	IF NOT arfbAlarm[4].bActive THEN
		arfbAlarm[4].Raise(nTimeStamp:=0);
	END_IF
	ELSE
	IF arfbAlarm[4].bActive AND GeneralAlarms.bReset THEN
		arfbAlarm[4].Clear(nTimeStamp:=0, bResetConfirmation:= FALSE);	
	END_IF	
// 	GeneralAlarms.bError:=TRUE;
// 	GeneralAlarms.bReset:=FALSE;
// 	GeneralAlarms.nErrorCode:=33;
// 	GeneralAlarms.udiStationID:=1;	
// 	GeneralAlarms.sStationName:='Błąd systemu';
// 	GeneralAlarms.sErrorString:='Błąd uruchamiania stacji | Brak możliwość wyłączenia stacji - zresetuj zasilanie';	
END_IF

//Alarm_0005	5	Error	Błąd bazowania | Zbyt długie bazowanie stacji - sprawdź urządzenia
// BLAD 34 - WatchDog stanu eResetting
IF TimerWatchdog_eResetting.Q  THEN
	IF NOT arfbAlarm[5].bActive THEN
		arfbAlarm[5].Raise(nTimeStamp:=0);
	END_IF
	ELSE
	IF arfbAlarm[5].bActive AND GeneralAlarms.bReset THEN
		arfbAlarm[5].Clear(nTimeStamp:=0, bResetConfirmation:= FALSE);	
	END_IF
// 	GeneralAlarms.bError:=TRUE;
// 	GeneralAlarms.bReset:=FALSE;
// 	GeneralAlarms.nErrorCode:=34;
// 	GeneralAlarms.udiStationID:=1;		
// 	GeneralAlarms.sStationName:='Błąd systemu';
// 	GeneralAlarms.sErrorString:='Błąd bazowania | Zbyt długie bazowanie stacji - sprawdź urządzenia';	
END_IF

//Alarm_0006	6	Error	Błąd zatrzymywania | Zbyt długie zatrzymywanie cyklu w trybie normalnym
// BLAD 35 - WatchDog stanu eStoping
IF TimerWatchdog_eStopping.Q (*AND NOT GeneralAlarms.bError*)  THEN
	IF NOT arfbAlarm[6].bActive THEN
		arfbAlarm[6].Raise(nTimeStamp:=0);
		P00_PackML.ACT_ResetCommands();
	END_IF
	ELSE
	IF arfbAlarm[6].bActive AND GeneralAlarms.bReset THEN
		arfbAlarm[6].Clear(nTimeStamp:=0, bResetConfirmation:= FALSE);	
	END_IF	
// 	GeneralAlarms.bError:=TRUE;
// 	GeneralAlarms.bReset:=FALSE;
// 	GeneralAlarms.bReset:=TRUE; {warning 'Dodany auto-reset przy błędzie nr 6'}	
// 	GeneralAlarms.nErrorCode:=35;
// 	GeneralAlarms.udiStationID:=1;	
// 	GeneralAlarms.sStationName:='Błąd systemu';
// 	GeneralAlarms.sErrorString:='Błąd zatrzymywania | Zbyt długie zatrzymywanie cyklu w trybie normalnym';	
END_IF

//Alarm_0007	7	Error	Błąd zasilania | Zanik fazy, lub zła kolejność faz - sprawdź podłączenie {0}	
//BŁĄD 36 - Zasilanie
IbLinearPowerSupplyOK;IbStepperPowerSupplyOK;IbStepperMotorsFuseOK;P07_ROPP.IbROPPFuseFB2OK;
IF 	(NOT IbPowerSupplyOK OR 
	(IbLinearPowerSupplyOK(*NCK*) AND tonEmergencyStop.Q) OR 
	(IbStepperPowerSupplyOK(*NOK*)AND tonEmergencyStop.Q) OR 
	(IbStepperMotorsFuseOK(*NOK*) AND tonEmergencyStop.Q) //OR 
	//(NOT P11_RollerScrewer.IbRollerScrewerFuseFB1OK AND tonEmergencyStop.Q)

	) THEN //AND (NOT P_Persistent.fbUPS_CU8130.stStatus.ePowerStatus=2) THEN//OR 
	//NOT IbFuse10F9OK OR NOT IbFuse10F11OK OR
	//NOT IbTurnTableOK OR NOT IbExitConveyorOK OR 
	//NOT P01_PucksInserter.IbPucksInserterFuseDrivesOK OR
	//NOT P01_PucksInserter.IbPucksInserterTransporter1OK OR
	//NOT P01_PucksInserter.IbPucksInserterTransporter2OK OR
	//NOT GVL_IO.IbPucksInserterRollerFuse OR	
	//NOT P01_PucksInserter.IbPucksInserterFuseFB1OK 	OR
	//NOT P07_ROPP.IbROPPFuseFB1OK OR 
	//(P07_ROPP.IbROPPFuseFB2OK (*NOK*) AND tonEmergencyStop.Q) AND
	//NOT P07_ROPP.IbROPPFuseFB3OK OR
	//NOT P07_ROPP.IbROPPFuseFB4OK OR
	//NOT P07_ROPP.IbROPPFuseFB5OK OR
	//NOT P07_ROPP.IbROPPFuseFB6OK OR 
	//NOT P07_ROPP.IbROPPFuseFB7OK OR
	//(NOT P07_ROPP.IbROPPFuseFB8OK AND tonEmergencyStop.Q)OR
	//(NOT P07_ROPP.IbROPPFuseFB9OK AND tonEmergencyStop.Q)
	VIS.bWritePersistent := TRUE;
// 	GeneralAlarms.bError:=TRUE;
// 	GeneralAlarms.bReset:=FALSE;
// 	GeneralAlarms.nErrorCode:=36;
// 	GeneralAlarms.udiStationID:=1;	
// 	GeneralAlarms.sStationName:='Błąd systemu';
// 	GeneralAlarms.sErrorString:='Błąd zasilania | Zanik fazy, lub zła kolejność faz - sprawdź podłączenie';
	sAlarmTest:='';
	IF NOT IbPowerSupplyOK THEN	sAlarmTest:=(*		GeneralAlarms.sErrorString2:=*)'R2-MainSupply';
	ELSIF NOT	P11_RollerScrewer.IbRollerScrewerFuseFB1OK  THEN sAlarmTest:=(*		GeneralAlarms.sErrorString2:=*)'RC40';
	//ELSIF IbLinearPowerSupplyOK THEN		GeneralAlarms.sErrorString2:='R2-LinearActuatorsSupply';
	//ELSIF IbStepperPowerSupplyOK THEN		GeneralAlarms.sErrorString2:='R2-StepperMotorsSupply';
	//ELSIF NOT IbFuseFanEXMotor THEN			GeneralAlarms.sErrorString2:='R2-FuseFanExSupply';	
	//ELSIF IbStepperMotorsFuseOK THEN		GeneralAlarms.sErrorString2:='R3-StepperMotorsFuse';
	//ELSIF NOT IbFuse10F9OK THEN				GeneralAlarms.sErrorString2:='R3-10F9';
	//ELSIF NOT IbFuse10F11OK THEN			GeneralAlarms.sErrorString2:='R3-10F11';
	//ELSIF NOT IbTurnTableOK THEN			GeneralAlarms.sErrorString2:='SO-TurnTable';
	//ELSIF NOT IbExitConveyorOK THEN			GeneralAlarms.sErrorString2:='SO-ExitConveyor';
	//ELSIF NOT P01_PucksInserter.IbPucksInserterFuseDrivesOK  THEN		GeneralAlarms.sErrorString2:='PI-71F1';
	//ELSIF NOT P01_PucksInserter.IbPucksInserterTransporter1OK  THEN		GeneralAlarms.sErrorString2:='PI-71F2';
	//ELSIF NOT P01_PucksInserter.IbPucksInserterTransporter2OK  THEN		GeneralAlarms.sErrorString2:='PI-71F3';
	//ELSIF NOT P01_PucksInserter.IbPucksInserterFuseFB1OK  THEN			GeneralAlarms.sErrorString2:='PI-10F15';
	//ELSIF NOT P07_ROPP.IbROPPFuseFB1OK  THEN							GeneralAlarms.sErrorString2:='ROPP-10F17';
	//ELSIF P07_ROPP.IbROPPFuseFB2OK  THEN								GeneralAlarms.sErrorString2:='ROPP-74M6-8';
	//ELSIF NOT P07_ROPP.IbROPPFuseFB3OK  THEN							GeneralAlarms.sErrorString2:='ROPP-74F6';
	//ELSIF NOT P07_ROPP.IbROPPFuseFB4OK  THEN							GeneralAlarms.sErrorString2:='ROPP-74F2';
	//ELSIF NOT P07_ROPP.IbROPPFuseFB5OK  THEN							GeneralAlarms.sErrorString2:='ROPP-74F3';
	//ELSIF NOT P07_ROPP.IbROPPFuseFB6OK  THEN							GeneralAlarms.sErrorString2:='ROPP-74F4';
	//ELSIF NOT P07_ROPP.IbROPPFuseFB7OK  THEN							GeneralAlarms.sErrorString2:='ROPP-74F5';
	//ELSIF NOT P07_ROPP.IbROPPFuseFB8OK  THEN							GeneralAlarms.sErrorString2:='ROPP-74F7';
	//ELSIF NOT P07_ROPP.IbROPPFuseFB9OK  THEN							GeneralAlarms.sErrorString2:='ROPP-74F7';		
	END_IF
	arfbAlarm[7].ipArguments.Clear() .AddString(sAlarmTest);
	IF NOT arfbAlarm[7].bActive THEN
		arfbAlarm[7].Raise(nTimeStamp:=0);
	END_IF
	ELSE	
	IF arfbAlarm[7].bActive AND GeneralAlarms.bReset THEN
		arfbAlarm[7].Clear(nTimeStamp:=0, bResetConfirmation:= FALSE);	
	END_IF		
	
END_IF	

//Alarm_0008	8	Error	Błąd zasilania DC | Alarm zasilacza 10G1 - sprawdź zasilanie
//BŁĄD 37 - Zasilanie DC
IF tonDCSupply1OK.Q THEN
//	VIS.bWritePersistent := TRUE;
	IF NOT arfbAlarm[8].bActive THEN
		IF  NOT P_Persistent.fbUPS_CU8130.stStatus.ePowerStatus=2 THEN
			VIS.bWritePersistent := TRUE;
		END_IF
		arfbAlarm[8].Raise(nTimeStamp:=0);
	END_IF
ELSE	
	IF arfbAlarm[8].bActive AND GeneralAlarms.bReset THEN
		arfbAlarm[8].Clear(nTimeStamp:=0, bResetConfirmation:= FALSE);	
	END_IF
// 	GeneralAlarms.bError:=TRUE;
// 	GeneralAlarms.bReset:=FALSE;
// 	GeneralAlarms.nErrorCode:=37;
// 	GeneralAlarms.udiStationID:=1;	
// 	GeneralAlarms.sStationName:='Błąd systemu';
// 	GeneralAlarms.sErrorString:='Błąd zasilania DC | Alarm zasilacza 10G1 - sprawdź zasilanie';
END_IF

//Alarm_0009	9	Error	Błąd zasilania DC | Alarm zasilacza 10G2 - sprawdź zasilanie	
//BŁĄD 38 - Zasilanie DC
IF (tonDCSupply2OK.Q  OR tonDCSupply3OK.Q) THEN
	IF NOT arfbAlarm[9].bActive THEN
		arfbAlarm[9].Raise(nTimeStamp:=0);
		IF NOT P_Persistent.fbUPS_CU8130.stStatus.ePowerStatus=2 THEN
		VIS.bWritePersistent := TRUE;
		END_IF
	END_IF
ELSE	
		IF arfbAlarm[9].bActive AND GeneralAlarms.bReset THEN
			arfbAlarm[9].Clear(nTimeStamp:=0, bResetConfirmation:= FALSE);	
		END_IF
//	VIS.bWritePersistent := TRUE;
// 	GeneralAlarms.bError:=TRUE;
// 	GeneralAlarms.bReset:=FALSE;
// 	GeneralAlarms.nErrorCode:=38;
// 	GeneralAlarms.udiStationID:=1;	
// 	GeneralAlarms.sStationName:='Błąd systemu';
// 	GeneralAlarms.sErrorString:='Błąd zasilania DC | Alarm zasilacza 10G2 - sprawdź zasilanie';
END_IF	

//Alarm_0010	10	Error	Błąd sprężonego powietrza | Zbyt niskie ciśnienie zasilania sprężonego powietrza - zwiększ ciśnienie {0}
//BŁĄD 39 - Zasilanie	
IF tonCompressedAir.Q THEN
// 	GeneralAlarms.bError:=TRUE;
// 	GeneralAlarms.bReset:=FALSE;
// 	GeneralAlarms.nErrorCode:=39;
// 	GeneralAlarms.udiStationID:=1;	
// 	GeneralAlarms.sStationName:='Błąd systemu';
// 	GeneralAlarms.sErrorString:='Błąd sprężonego powietrza | Zbyt niskie ciśnienie zasilania sprężonego powietrza - zwiększ ciśnienie';
	IF NOT IbCompressedAirOK AND IbEmergencyStop THEN
		GeneralAlarms.sErrorString2:='UL';
	//ELSIF NOT P07_ROPP.IbROPPCompressedAirOK THEN
	//	GeneralAlarms.sErrorString2:='ROPP';
	END_IF
	arfbAlarm[10].ipArguments.Clear() .AddString(GeneralAlarms.sErrorString2);
	IF NOT arfbAlarm[10].bActive THEN
		arfbAlarm[10].Raise(nTimeStamp:=0);
	END_IF
	ELSE	
	IF arfbAlarm[10].bActive AND GeneralAlarms.bReset THEN
		arfbAlarm[10].Clear(nTimeStamp:=0, bResetConfirmation:= FALSE);	
	END_IF
END_IF

//Alarm_0011	11	Error	Błąd bezpieczników 24VDC | Jeden z bezpieczników w bloku FB1 uległ przepaleniu - wymień bezpiecznik
//BŁĄD 40 - przepalony bezpiecznik FB1
IF tonFuseFB1OK.Q THEN
	IF NOT arfbAlarm[11].bActive THEN
		arfbAlarm[11].Raise(nTimeStamp:=0);
	END_IF
	ELSE	
	IF arfbAlarm[11].bActive AND GeneralAlarms.bReset THEN
		arfbAlarm[11].Clear(nTimeStamp:=0, bResetConfirmation:= FALSE);	
	END_IF
// 	GeneralAlarms.bError:=TRUE;
// 	GeneralAlarms.bReset:=FALSE;
// 	GeneralAlarms.nErrorCode:=40;
// 	GeneralAlarms.udiStationID:=1;	
// 	GeneralAlarms.sStationName:='Błąd systemu';
// 	GeneralAlarms.sErrorString:='Błąd bezpieczników 24VDC | Jeden z bezpieczników w bloku FB1 uległ przepaleniu - wymień bezpiecznik';
END_IF

//Alarm_0012	12	Error	Błąd bezpieczników 24VDC | Jeden z bezpieczników w bloku FB2 uległ przepaleniu - wymień bezpiecznik
//BŁĄD 41 - przepalony bezpiecznik FB2	zrobic timer
IF tonFuseFB2OK.Q THEN
	IF NOT arfbAlarm[12].bActive THEN
		arfbAlarm[12].Raise(nTimeStamp:=0);
	END_IF
	ELSE	
	IF arfbAlarm[12].bActive AND GeneralAlarms.bReset THEN
		arfbAlarm[12].Clear(nTimeStamp:=0, bResetConfirmation:= FALSE);	
	END_IF
// 	GeneralAlarms.bError:=TRUE;
// 	GeneralAlarms.bReset:=FALSE;
// 	GeneralAlarms.nErrorCode:=41;
// 	GeneralAlarms.udiStationID:=1;	
// 	GeneralAlarms.sStationName:='Błąd systemu';
// 	GeneralAlarms.sErrorString:='Błąd bezpieczników 24VDC | Jeden z bezpieczników w bloku FB2 uległ przepaleniu - wymień bezpiecznik';
END_IF

//Alarm_0013	13	Error	Błąd bezpieczników 24VDC | Jeden z bezpieczników w bloku FB3 uległ przepaleniu - wymień bezpiecznik
//BŁĄD 42 - przepalony bezpiecznik FB3	
(*ELSIF tonFuseFB3OK.Q THEN
	GeneralAlarms.bError:=TRUE;
	GeneralAlarms.bReset:=FALSE;
	GeneralAlarms.nErrorCode:=42;
	GeneralAlarms.udiStationID:=1;	
	GeneralAlarms.sStationName:='Błąd systemu';
	GeneralAlarms.sErrorString:='Błąd bezpieczników 24VDC | Jeden z bezpieczników w bloku FB3 uległ przepaleniu - wymień bezpiecznik';*)

//Alarm_0014	14	Error	Serwowzmacniacz | Wyłączone zabezpieczenie silnikowe - sprawdż zabezpieczenie
//BŁĄD 43 - zabezpieczenie silnikowe napęd transportera
IF NOT IbFuseDrivesOK THEN
	IF NOT arfbAlarm[14].bActive THEN
		arfbAlarm[14].Raise(nTimeStamp:=0);
	END_IF
	ELSE	
	IF arfbAlarm[14].bActive AND GeneralAlarms.bReset THEN
		arfbAlarm[14].Clear(nTimeStamp:=0, bResetConfirmation:= FALSE);	
	END_IF
// 	GeneralAlarms.bError:=TRUE;
// 	GeneralAlarms.bReset:=FALSE;
// 	GeneralAlarms.nErrorCode:=43;
// 	GeneralAlarms.udiStationID:=1;	
// 	GeneralAlarms.sStationName:='Błąd systemu';
// 	GeneralAlarms.sErrorString:='Serwowzmacniacz | Wyłączone zabezpieczenie silnikowe - sprawdż zabezpieczenie';
END_IF
	
(**//Alarm_0015	15	Error	Napęd transportera | Wyłączone zabezpieczenie silnikowe - sprawdż zabezpieczenie
//BŁĄD 44 - zabezpieczenie silnikowe napęd transportera
IF NOT IbFuseFormTransporter1OK THEN
	IF NOT arfbAlarm[15].bActive THEN
		arfbAlarm[15].Raise(nTimeStamp:=0);
	END_IF
	ELSE	
	IF arfbAlarm[15].bActive AND GeneralAlarms.bReset THEN
		arfbAlarm[15].Clear(nTimeStamp:=0, bResetConfirmation:= FALSE);	
	END_IF
// 	GeneralAlarms.bError:=TRUE;
// 	GeneralAlarms.bReset:=FALSE;
// 	GeneralAlarms.nErrorCode:=44;
// 	GeneralAlarms.udiStationID:=1;	
// 	GeneralAlarms.sStationName:='Błąd systemu';
// 	GeneralAlarms.sErrorString:='Napęd transportera | Wyłączone zabezpieczenie silnikowe - sprawdż zabezpieczenie';
END_IF	*)

//Alarm_0016	16	Error	Napęd obrotu stacji znakowania | Wyłączone zabezpieczenie silnikowe - sprawdż zabezpieczenie
//BŁĄD 45 - zabezpieczenie silnikowe napędu injketowania obwodowego
IF NOT IbFuseCircularInkjetOK AND bCircularInkjetEnable THEN
	IF NOT arfbAlarm[16].bActive THEN
		arfbAlarm[16].Raise(nTimeStamp:=0);
	END_IF
	ELSE	
	IF arfbAlarm[16].bActive AND GeneralAlarms.bReset THEN
		arfbAlarm[16].Clear(nTimeStamp:=0, bResetConfirmation:= FALSE);	
	END_IF
// 	GeneralAlarms.bError:=TRUE;
// 	GeneralAlarms.bReset:=FALSE;
// 	GeneralAlarms.nErrorCode:=45;
// 	GeneralAlarms.udiStationID:=1;	
// 	GeneralAlarms.sStationName:='Błąd systemu';
// 	GeneralAlarms.sErrorString:='Napęd obrotu stacji znakowania | Wyłączone zabezpieczenie silnikowe - sprawdż zabezpieczenie';
END_IF	

//Alarm_0017	17	Error	Stacja wyjściowa | Niewyjęta butelka z formatki - usuń butelkę
//BŁĄD 46 - Niewyjęta butelka przez robota - usuń butelkę																			
IF tonBottleCheckAfterBottleTransferSensor.Q  THEN
	IF NOT arfbAlarm[17].bActive THEN
		arfbAlarm[17].Raise(nTimeStamp:=0);
	END_IF
	ELSE	
	IF arfbAlarm[17].bActive AND GeneralAlarms.bReset THEN
		arfbAlarm[17].Clear(nTimeStamp:=0, bResetConfirmation:= FALSE);	
	END_IF
// 	GeneralAlarms.bError:=TRUE;
// 	GeneralAlarms.bReset:=FALSE;
// 	GeneralAlarms.nErrorCode:=46;
// 	GeneralAlarms.udiStationID:=1;	
// 	GeneralAlarms.sStationName:='Błąd systemu';// ąśźżłóćęŁĄĆŚŻŹ¹';
// 	GeneralAlarms.sErrorString:='Stacja wyjściowa | Niewyjęta butelka z formatki - usuń butelkę'; //ąśźżłóćęŁĄĆŚŻŹ¹';
END_IF	

//Alarm_0018	18	Error	Stacja wejściowa | Źle włozona butelka - popraw
//BŁĄD 47 - Źle włozona butelka - popraw																		
IF tonIbBottleNotInserted.Q  THEN
	IF NOT arfbAlarm[18].bActive THEN
		arfbAlarm[18].Raise(nTimeStamp:=0);
	END_IF
	ELSE	
	IF arfbAlarm[18].bActive AND GeneralAlarms.bReset THEN
		arfbAlarm[18].Clear(nTimeStamp:=0, bResetConfirmation:= FALSE);	
	END_IF
// 	GeneralAlarms.bError:=TRUE;
// 	GeneralAlarms.bReset:=FALSE;
// 	GeneralAlarms.nErrorCode:=47;
// 	GeneralAlarms.udiStationID:=1;	
// 	GeneralAlarms.sStationName:='Błąd systemu';
// 	GeneralAlarms.sErrorString:='Stacja wejściowa | Źle włozona butelka - popraw';
END_IF	

//Alarm_0019	19	Error	Sterownik główny | Brak napięcia zasilania na module ST2 w szafie głównej - sprawdź bezpiecznik
//BŁĄD 48 - Brak napięcia zasilania na module ST1 w szafie głównej		
IF tonPowerSuppyTerminal1UsUndervoltageError.Q THEN
	IF NOT arfbAlarm[19].bActive THEN
		arfbAlarm[19].Raise(nTimeStamp:=0);
	END_IF
	ELSE	
	IF arfbAlarm[19].bActive AND GeneralAlarms.bReset THEN
		arfbAlarm[19].Clear(nTimeStamp:=0, bResetConfirmation:= FALSE);	
	END_IF
// 	GeneralAlarms.bError:=TRUE;
// 	GeneralAlarms.bReset:=FALSE;
// 	GeneralAlarms.nErrorCode:=48;
// 	GeneralAlarms.udiStationID:=1;	
// 	GeneralAlarms.sStationName:='Błąd systemu';
// 	GeneralAlarms.sErrorString:='Sterownik główny | Brak napięcia zasilania na module ST2 w szafie głównej - sprawdź bezpiecznik';
END_IF	

//Alarm_0020	20	Error	Sterownik w szafie robota | Brak napięcia zasilania na module ST1 w szafie robota - sprawdź bezpiecznik
//BŁĄD 49 - Brak napięcia zasilania na module ST1 w szafie robota
IF tonPowerSuppyTerminal2UpUndervoltageError.Q THEN
	IF NOT arfbAlarm[20].bActive THEN
		arfbAlarm[20].Raise(nTimeStamp:=0);
	END_IF
	ELSE	
	IF arfbAlarm[20].bActive AND GeneralAlarms.bReset THEN
		arfbAlarm[20].Clear(nTimeStamp:=0, bResetConfirmation:= FALSE);	
	END_IF
// 	GeneralAlarms.bError:=TRUE;
// 	GeneralAlarms.bReset:=FALSE;
// 	GeneralAlarms.nErrorCode:=49;
// 	GeneralAlarms.udiStationID:=1;	
// 	GeneralAlarms.sStationName:='Błąd systemu';
// 	GeneralAlarms.sErrorString:='Sterownik w szafie robota | Brak napięcia zasilania na module ST1 w szafie robota - sprawdź bezpiecznik';
END_IF	

//Alarm_0021	21	Error	Sterownik w szafie robota | Brak napięcia E-Bus na module ST1 w szafie robota - sprawdź bezpiecznik
//BŁĄD 50 - Brak napięcia E-Bus na module ST1 w szafie robota		
IF tonPowerSuppyTerminal2UsUndervoltageError.Q THEN
	IF NOT arfbAlarm[21].bActive THEN
		arfbAlarm[21].Raise(nTimeStamp:=0);
	END_IF
	ELSE	
	IF arfbAlarm[21].bActive AND GeneralAlarms.bReset THEN
		arfbAlarm[21].Clear(nTimeStamp:=0, bResetConfirmation:= FALSE);	
	END_IF
// 	GeneralAlarms.bError:=TRUE;
// 	GeneralAlarms.bReset:=FALSE;
// 	GeneralAlarms.nErrorCode:=50;
// 	GeneralAlarms.udiStationID:=1;	
// 	GeneralAlarms.sStationName:='Błąd systemu';
// 	GeneralAlarms.sErrorString:='Sterownik w szafie robota | Brak napięcia E-Bus na module ST1 w szafie robota - sprawdź bezpiecznik';
END_IF

//Alarm_0022	22	Error	Stacja zakręcarek | Zablokowana formatka za zakręcarką sprawdź położenie
//BŁĄD 51 -	Zablokowana formatka przy stacji zakręcarek
IF tonFormsStuckAfterScrewersAlarm.Q  THEN
	IF NOT arfbAlarm[22].bActive THEN
		arfbAlarm[22].Raise(nTimeStamp:=0);
	END_IF
	ELSE	
	IF arfbAlarm[22].bActive AND GeneralAlarms.bReset THEN
		arfbAlarm[22].Clear(nTimeStamp:=0, bResetConfirmation:= FALSE);	
	END_IF
// 	GeneralAlarms.bError:=TRUE;
// 	GeneralAlarms.bReset:=FALSE;
// 	GeneralAlarms.nErrorCode:=51;
// 	GeneralAlarms.udiStationID:=1;	
// 	GeneralAlarms.sStationName:='Błąd systemu';
// 	GeneralAlarms.sErrorString:='Stacja zakręcarek | Zablokowana formatka za zakręcarką sprawdź położenie';
END_IF

(*//Alarm_0023	23	Error	Napęd transportera | Wyłączone zabezpieczenie silnikowe - sprawdż zabezpieczenie			aGeneralAlarms				
//BŁĄD 52 - zabezpieczenie silnikowe napęd transportera
IF NOT IbFuseFormTransporter2OK THEN
	IF NOT arfbAlarm[23].bActive THEN
		arfbAlarm[23].Raise(nTimeStamp:=0);
	END_IF
	ELSE	
	IF arfbAlarm[23].bActive AND GeneralAlarms.bReset THEN
		arfbAlarm[23].Clear(nTimeStamp:=0, bResetConfirmation:= FALSE);	
	END_IF
// 	GeneralAlarms.bError:=TRUE;
// 	GeneralAlarms.bReset:=FALSE;
// 	GeneralAlarms.nErrorCode:=52;
// 	GeneralAlarms.udiStationID:=1;	
// 	GeneralAlarms.sStationName:='Błąd systemu';
// 	GeneralAlarms.sErrorString:='Napęd transportera | Wyłączone zabezpieczenie silnikowe - sprawdż zabezpieczenie';
END_IF	

//Alarm_0024	24	Error	Napęd transportera | Wyłączone zabezpieczenie silnikowe - sprawdż zabezpieczenie
//BŁĄD 53 - zabezpieczenie silnikowe napęd transportera
IF NOT IbFuseFormTransporter3OK THEN
	IF NOT arfbAlarm[24].bActive THEN
		arfbAlarm[24].Raise(nTimeStamp:=0);
	END_IF
	ELSE	
	IF arfbAlarm[24].bActive AND GeneralAlarms.bReset THEN
		arfbAlarm[24].Clear(nTimeStamp:=0, bResetConfirmation:= FALSE);	
	END_IF
// 	GeneralAlarms.bReset:=FALSE;
// 	GeneralAlarms.nErrorCode:=53;
// 	GeneralAlarms.udiStationID:=1;	
// 	GeneralAlarms.sStationName:='Błąd systemu';
// 	GeneralAlarms.sErrorString:='Napęd transportera | Wyłączone zabezpieczenie silnikowe - sprawdż zabezpieczenie';
END_IF	

//Alarm_0025	25	Error	Napęd transportera | Wyłączone zabezpieczenie silnikowe - sprawdż zabezpieczenie 
//BŁĄD 54 - zabezpieczenie silnikowe napęd transportera
IF (NOT IbFuseFormTransporter4OK OR NOT IbFuseFormTransporter5OK) THEN
	IF NOT arfbAlarm[25].bActive THEN
		arfbAlarm[25].Raise(nTimeStamp:=0);
	END_IF
	ELSE	
	IF arfbAlarm[25].bActive AND GeneralAlarms.bReset THEN
		arfbAlarm[25].Clear(nTimeStamp:=0, bResetConfirmation:= FALSE);	
	END_IF
// 	GeneralAlarms.bError:=TRUE;
// 	GeneralAlarms.bReset:=FALSE;
// 	GeneralAlarms.nErrorCode:=54;
// 	GeneralAlarms.udiStationID:=1;	
// 	GeneralAlarms.sStationName:='Błąd systemu';
// 	GeneralAlarms.sErrorString:='Napęd transportera | Wyłączone zabezpieczenie silnikowe - sprawdż zabezpieczenie';
END_IF	
	
//Alarm_0026	26	Error	Napęd transportera | Wyłączone zabezpieczenie silnikowe - sprawdż zabezpieczenie
//BŁĄD 55 - zabezpieczenie silnikowe napęd transportera
IF NOT IbFuseFormTransporter4OK THEN
	IF NOT arfbAlarm[26].bActive THEN
		arfbAlarm[26].Raise(nTimeStamp:=0);
	END_IF
	ELSE	
	IF arfbAlarm[26].bActive AND GeneralAlarms.bReset THEN
		arfbAlarm[26].Clear(nTimeStamp:=0, bResetConfirmation:= FALSE);	
	END_IF
// 	GeneralAlarms.bError:=TRUE;
// 	GeneralAlarms.bReset:=FALSE;
// 	GeneralAlarms.nErrorCode:=55;
// 	GeneralAlarms.udiStationID:=1;	
// 	GeneralAlarms.sStationName:='Błąd systemu';
// 	GeneralAlarms.sErrorString:='Napęd transportera | Wyłączone zabezpieczenie silnikowe - sprawdż zabezpieczenie';
END_IF*)

//Alarm_0027	27	Error	Napęd stołu obrotowego | Wyłączone zabezpieczenie silnikowe - sprawdż zabezpieczenie
//BŁĄD 56  - zabezpieczenie silnikowe napęd stołu obrotowego
//ELSIF (NOT IbBottleFeederTurntableOK AND bBottleFeederEnable) THEN
//	GeneralAlarms.bError:=TRUE;
//	GeneralAlarms.bReset:=FALSE;
//	GeneralAlarms.nErrorCode:=56;
//	GeneralAlarms.udiStationID:=1;	
//	GeneralAlarms.sStationName:='Błąd systemu';
//	GeneralAlarms.sErrorString:='Napęd stołu obrotowego | Wyłączone zabezpieczenie silnikowe - sprawdż zabezpieczenie';

//Alarm_0028	28	Error	Transporter odrzuconych | Zapełniony transporter odrzuconych butelek
//Błąd 57 zapełniony transporter odrzuconych 
IF tonBadBottleConvoyerAlarm.Q THEN
	IF NOT arfbAlarm[28].bActive THEN
		arfbAlarm[28].Raise(nTimeStamp:=0);
	END_IF
	ELSE	
	IF arfbAlarm[28].bActive AND GeneralAlarms.bReset THEN
		arfbAlarm[28].Clear(nTimeStamp:=0, bResetConfirmation:= FALSE);	
	END_IF
// 	GeneralAlarms.bError:=TRUE;
// 	GeneralAlarms.bReset:=FALSE;
// 	GeneralAlarms.nErrorCode:=57;
// 	GeneralAlarms.udiStationID:=1;	
// 	GeneralAlarms.sStationName:='Błąd systemu';
// 	GeneralAlarms.sErrorString:='Transporter odrzuconych | Zapełniony transporter odrzuconych butelek';
END_IF	

//Alarm_0029	29	Error	Stacja dozowników | Zablokowana formatka przy dozownikach od strony drzwi. Usuń formatki i opakowania
//Błąd 58 zablokowana formatka przy dozownikach
IF tonFormStuckAfterDispencer34Alarm.Q AND VIS.bDosingTwoPhasesShow THEN
	IF NOT arfbAlarm[29].bActive THEN
		arfbAlarm[29].Raise(nTimeStamp:=0);
	END_IF
	ELSE	
	IF arfbAlarm[29].bActive AND GeneralAlarms.bReset THEN
		arfbAlarm[29].Clear(nTimeStamp:=0, bResetConfirmation:= FALSE);	
	END_IF
// 	GeneralAlarms.bError:=TRUE;
// 	GeneralAlarms.bReset:=FALSE;
// 	GeneralAlarms.nErrorCode:=58;
// 	GeneralAlarms.udiStationID:=1;	
// 	GeneralAlarms.sStationName:='Błąd systemu';
// 	GeneralAlarms.sErrorString:='Stacja dozowników | Zablokowana formatka przy dozownikach od strony drzwi. Usuń formatki i opakowania';
END_IF

//Alarm_0030	30	Error	Stacja zakręcarek | Zablokowana lub źle ustawiona formatka przed zakręcarkami. Sprawdź ustawienie formatek oraz czujniki obecności
//Błąd 59 zablokowanej formatki przed zakręcarkmi
IF tonbFormsStuckBeforeScrewersAlarm.Q THEN
	IF NOT arfbAlarm[30].bActive THEN
		arfbAlarm[30].Raise(nTimeStamp:=0);
	END_IF
	ELSE	
	IF arfbAlarm[30].bActive AND GeneralAlarms.bReset THEN
		arfbAlarm[30].Clear(nTimeStamp:=0, bResetConfirmation:= FALSE);	
	END_IF
// 	GeneralAlarms.bError:=TRUE;
// 	GeneralAlarms.bReset:=FALSE;
// 	GeneralAlarms.nErrorCode:=59;
// 	GeneralAlarms.udiStationID:=1;	
// 	GeneralAlarms.sStationName:='Błąd systemu';
// 	GeneralAlarms.sErrorString:='Stacja zakręcarek | Zablokowana lub źle ustawiona formatka przed zakręcarkami. Sprawdź ustawienie formatek oraz czujniki obecności';
END_IF

//Alarm_0031	31	Error	Stacja zakręcarek | Źle ustawione formatki przed zakręcarką. Sprawdź czujniki obecności formatek
//Błąd 60 zablokowanej formatki przed zakręcarkmi
IF tonFormsStuckBeforeScrewersAlarm2.Q THEN
	IF NOT arfbAlarm[31].bActive THEN
		arfbAlarm[31].Raise(nTimeStamp:=0);
	END_IF
	ELSE	
	IF arfbAlarm[31].bActive AND GeneralAlarms.bReset THEN
		arfbAlarm[31].Clear(nTimeStamp:=0, bResetConfirmation:= FALSE);	
	END_IF
// 	GeneralAlarms.bError:=TRUE;
// 	GeneralAlarms.bReset:=FALSE;
// 	GeneralAlarms.nErrorCode:=60;
// 	GeneralAlarms.udiStationID:=1;	
// 	GeneralAlarms.sStationName:='Błąd systemu';
// 	GeneralAlarms.sErrorString:='Stacja zakręcarek | Źle ustawione formatki przed zakręcarką. Sprawdź czujniki obecności formatek';
END_IF

//Alarm_0032	32	Error	Stacja dozowników |Źle ustawione formatki przy dozownikach od strony drzwi. Przesuń formatki za wagi
//Błąd 61 zablokowanej formatki za dozownikami
IF tonFormStuckAfterDispencerAlarm.Q THEN
	IF NOT arfbAlarm[32].bActive THEN
		arfbAlarm[32].Raise(nTimeStamp:=0);
	END_IF
	ELSE	
	IF arfbAlarm[32].bActive AND GeneralAlarms.bReset THEN
		arfbAlarm[32].Clear(nTimeStamp:=0, bResetConfirmation:= FALSE);	
	END_IF
// 	GeneralAlarms.bError:=TRUE;
// 	GeneralAlarms.bReset:=FALSE;
// 	GeneralAlarms.nErrorCode:=61;
// 	GeneralAlarms.sStationName:='Błąd systemu';
// 	GeneralAlarms.sErrorString:='Stacja dozowników | Źle ustawione formatki przy dozownikach od strony drzwi. Przesuń formatki za wagi';
END_IF

//Alarm_0033	33	Error	Podajnik zamknięć | Brak zamknięć w 8 butelkach - sprawdź sorter
//BŁĄD 62 - Brak nasadek po sorterze 
//wykomentowany błąd 8 butelek
IF (iCapFeederCheckCountNOK >= 3 AND bCapFeederEnable) THEN  //stCapSorterRead.bEnable AND NOT bCapSorterDisable) THEN
	IF NOT arfbAlarm[33].bActive THEN
		arfbAlarm[33].Raise(nTimeStamp:=0);
	END_IF
	ELSE	
	IF arfbAlarm[33].bActive AND GeneralAlarms.bReset THEN
		arfbAlarm[33].Clear(nTimeStamp:=0, bResetConfirmation:= FALSE);	
	END_IF
// 	GeneralAlarms.bError:=TRUE;
// 	GeneralAlarms.bReset:=FALSE;
// 	GeneralAlarms.nErrorCode:=62;
// 	GeneralAlarms.udiStationID:=1;	
// 	GeneralAlarms.sStationName:='Błąd systemu';
// 	GeneralAlarms.sErrorString:='Podajnik zamknięć | Brak zamknięć w 8 butelkach - sprawdź sorter';
END_IF

//Alarm_0034	34	Error	Brak gotowości stacji | Zbyt długie przygotowywanie stacji do gotowości
// BLAD 63 - WatchDog stanu Idle ale bez gotowych stacji
IF TimerWatchdog_eIdleAndNotStationsAreReady.Q AND (IbCycleStartButton OR IbTurnTableCycleStartButton OR P07_ROPP.IbROPPCycleStartButton)  THEN
// 	GeneralAlarms.bError:=TRUE;
// 	GeneralAlarms.bReset:=FALSE;
// 	GeneralAlarms.nErrorCode:=63;
// 	GeneralAlarms.udiStationID:=1;	
// 	GeneralAlarms.sStationName:='Błąd systemu';
// 	GeneralAlarms.sErrorString:='Brak gotowości stacji | Zbyt długie przygotowywanie stacji do gotowości';
	GeneralAlarms.sErrorString2:='';
	IF P01_BottleFeeder.fbBottleFeeder.eState <> E_Station.eReady AND bBottleFeederEnable THEN
		GeneralAlarms.sErrorString2:='Round bottle inserter';		
	END_IF
	arfbAlarm[34].ipArguments.Clear() .AddString(GeneralAlarms.sErrorString2);
	IF NOT arfbAlarm[34].bActive THEN
		arfbAlarm[34].Raise(nTimeStamp:=0);
	END_IF
	ELSE	
	IF arfbAlarm[34].bActive AND GeneralAlarms.bReset THEN
		arfbAlarm[34].Clear(nTimeStamp:=0, bResetConfirmation:= FALSE);	
	END_IF
END_IF

//Alarm_0035	35	Error	Stacja zakręcarek | Formatki nie są dosunięte do pozycji przeciągania - odblokuj (wypadła nakrętka)
//Błąd 64 wypadła nakretka przez zakrecarką
IF tonFormsStuckBeforeScrewersAlarm3.Q THEN
	IF NOT arfbAlarm[35].bActive THEN
		arfbAlarm[35].Raise(nTimeStamp:=0);
	END_IF
	ELSE	
	IF arfbAlarm[35].bActive AND GeneralAlarms.bReset THEN
		arfbAlarm[35].Clear(nTimeStamp:=0, bResetConfirmation:= FALSE);	
	END_IF
// 	GeneralAlarms.bError:=TRUE;
// 	GeneralAlarms.bReset:=FALSE;
// 	GeneralAlarms.nErrorCode:=64;
// 	GeneralAlarms.udiStationID:=1;	
// 	GeneralAlarms.sStationName:='Błąd systemu';
// 	GeneralAlarms.sErrorString:='Stacja zakręcarek | Formatki nie są dosunięte do pozycji przeciągania - odblokuj (wypadła nakrętka)';
END_IF	

//Alarm_0036	36	Error	Sorter butelek | Brak komunikacji ze sterownikiem - włącz zasilanie/sprawdź podłączenie
//Błąd 65 brak komunikacji ze sterownikiem sortera butelek
IF tonstBottleSorterReadiWatchdog.Q THEN
	IF NOT arfbAlarm[36].bActive THEN
		arfbAlarm[36].Raise(nTimeStamp:=0);
	END_IF
	ELSE	
	IF arfbAlarm[36].bActive AND GeneralAlarms.bReset THEN
		arfbAlarm[36].Clear(nTimeStamp:=0, bResetConfirmation:= FALSE);	
	END_IF
// 	GeneralAlarms.bError:=TRUE;
// 	GeneralAlarms.bReset:=FALSE;
// 	GeneralAlarms.nErrorCode:=65;
// 	GeneralAlarms.udiStationID:=1;	
// 	GeneralAlarms.sStationName:='Błąd systemu';
// 	GeneralAlarms.sErrorString:='Sorter butelek | Brak komunikacji ze sterownikiem - włącz zasilanie/sprawdź podłączenie';
END_IF	

//Alarm_0037	37	Error	Sorter nasadek | Brak komunikacji ze sterownikiem - włącz zasilanie/sprawdź podłączenie
//Błąd 66 brak komunikacji ze sterownikiem sortera nasadek
IF tonstBottleSorterReadiWatchdog.Q THEN
	IF NOT arfbAlarm[37].bActive THEN
		arfbAlarm[37].Raise(nTimeStamp:=0);
	END_IF
	ELSE	
	IF arfbAlarm[37].bActive AND GeneralAlarms.bReset THEN
		arfbAlarm[37].Clear(nTimeStamp:=0, bResetConfirmation:= FALSE);	
	END_IF
// 	GeneralAlarms.bError:=TRUE;
// 	GeneralAlarms.bReset:=FALSE;
// 	GeneralAlarms.nErrorCode:=66;
// 	GeneralAlarms.udiStationID:=1;	
// 	GeneralAlarms.sStationName:='Błąd systemu';
// 	GeneralAlarms.sErrorString:='Sorter nasadek | Brak komunikacji ze sterownikiem - włącz zasilanie/sprawdź podłączenie';
END_IF	

//Alarm_0038	38	Error	Sorter nasadek - przeciąganie | Formatki nie są dosunięte do pozycji przeciągania - odblokuj (wypadła nakrętka)
//Błąd 67 wypadła nakretka przed sorterem nakretek
IF tonFormsStuckBeforeCapSorterAlarm.Q THEN
	IF NOT arfbAlarm[38].bActive THEN
		arfbAlarm[38].Raise(nTimeStamp:=0);
	END_IF
	ELSE	
	IF arfbAlarm[38].bActive AND GeneralAlarms.bReset THEN
		arfbAlarm[38].Clear(nTimeStamp:=0, bResetConfirmation:= FALSE);	
	END_IF
// 	GeneralAlarms.bError:=TRUE;
// 	GeneralAlarms.bReset:=FALSE;
// 	GeneralAlarms.nErrorCode:=67;
// 	GeneralAlarms.udiStationID:=1;	
// 	GeneralAlarms.sStationName:='Błąd systemu';
// 	GeneralAlarms.sErrorString:='Sorter nasadek - przeciąganie | Formatki nie są dosunięte do pozycji przeciągania - odblokuj (wypadła nakrętka)';	
END_IF

//Alarm_0039	39	Error	Układ bezpieczeństwa | Brak komunikacji z sorterem nasadek - włącz linie/sprawdź komunikacje
IF IbCommunicationErrorUF50 AND IbEmergencyStop AND P00_PackML.tonbFirstCycle.Q THEN
	IF NOT arfbAlarm[39].bActive THEN
		arfbAlarm[39].Raise(nTimeStamp:=0);
	END_IF
	ELSE	
	IF arfbAlarm[39].bActive AND GeneralAlarms.bReset THEN
		arfbAlarm[39].Clear(nTimeStamp:=0, bResetConfirmation:= FALSE);	
	END_IF
// 	GeneralAlarms.bError:=TRUE;
// 	GeneralAlarms.bReset:=FALSE;
// 	GeneralAlarms.nErrorCode:=68;
// 	GeneralAlarms.udiStationID:=1;	
// 	GeneralAlarms.sStationName:='Błąd systemu';
// 	GeneralAlarms.sErrorString:='Układ bezpieczeństwa | Brak komunikacji z sorterem nasadek - włącz linie/sprawdź komunikacje';	
END_IF	

//Alarm_0040	40	Error	Układ bezpieczeństwa | Brak komunikacji z sorterem butelek - włącz linie/sprawdź komunikacje
//Błąd 69 bład komunikacji safety z sorterem butelek
IF IbCommunicationErrorUP50B AND IbEmergencyStop AND P00_PackML.tonbFirstCycle.Q THEN
	IF NOT arfbAlarm[40].bActive THEN
		arfbAlarm[40].Raise(nTimeStamp:=0);
	END_IF
	ELSE	
	IF arfbAlarm[40].bActive AND GeneralAlarms.bReset THEN
		arfbAlarm[40].Clear(nTimeStamp:=0, bResetConfirmation:= FALSE);	
	END_IF
// 	GeneralAlarms.bError:=TRUE;
// 	GeneralAlarms.bReset:=FALSE;
// 	GeneralAlarms.nErrorCode:=69;
// 	GeneralAlarms.udiStationID:=1;	
// 	GeneralAlarms.sStationName:='Błąd systemu';
// 	GeneralAlarms.sErrorString:='Układ bezpieczeństwa | Brak komunikacji z sorterem butelek - włącz linie/sprawdź komunikacje';	
END_IF	

//Alarm_0041	41	Error	Stacja dozowników | Formatki nie są dosunięte do pozycji przeciągania - odblokuj (wypadła butelka)
//Błąd 70 wypadła butelka przed dozownikami
IF tonFormStuckBeforeDispencer14Alarm.Q THEN
	IF NOT arfbAlarm[41].bActive THEN
		arfbAlarm[41].Raise(nTimeStamp:=0);
	END_IF
	ELSE	
	IF arfbAlarm[41].bActive AND GeneralAlarms.bReset THEN
		arfbAlarm[41].Clear(nTimeStamp:=0, bResetConfirmation:= FALSE);	
	END_IF
// 	GeneralAlarms.bError:=TRUE;
// 	GeneralAlarms.bReset:=FALSE;
// 	GeneralAlarms.nErrorCode:=70;
// 	GeneralAlarms.udiStationID:=1;	
// 	GeneralAlarms.sStationName:='Błąd systemu';
// 	GeneralAlarms.sErrorString:='Stacja dozowników | Formatki nie są dosunięte do pozycji przeciągania - odblokuj (wypadła butelka)';	
END_IF	

//Alarm_0042	42	Error	Napęd stołu odbiorczego | Wyłączone zabezpieczenie silnikowe - sprawdż zabezpieczenie
//BŁĄD 71  - zabezpieczenie silnikowe napęd stołu odbiorczego
//ELSIF (NOT IbTurnTableOK AND bExitTurnTableEnable) THEN
//	GeneralAlarms.bError:=TRUE;
//	GeneralAlarms.bReset:=FALSE;
//	GeneralAlarms.nErrorCode:=71;
//	GeneralAlarms.udiStationID:=1;	
//	GeneralAlarms.sStationName:='Błąd systemu';
//	GeneralAlarms.sErrorString:='Napęd stołu odbiorczego | Wyłączone zabezpieczenie silnikowe - sprawdż zabezpieczenie';
	
//Alarm_0043	43	Error	Stacja przeciągania dozowniki lewe | Pozycja podnośnika dozowników jest poniżej ustawionej
//BŁĄD 80  	
IF tonbFormsDragingLeftRunCheck.Q THEN
	IF NOT arfbAlarm[43].bActive THEN
		arfbAlarm[43].Raise(nTimeStamp:=0);
	END_IF
	ELSE	
	IF arfbAlarm[43].bActive AND GeneralAlarms.bReset THEN
		arfbAlarm[43].Clear(nTimeStamp:=0, bResetConfirmation:= FALSE);	
	END_IF
// 	GeneralAlarms.bError:=TRUE;
// 	GeneralAlarms.bReset:=FALSE;
// 	GeneralAlarms.nErrorCode:=80;
// 	GeneralAlarms.sStationName:='Stacja przeciągania dozowniki lewe';
// 	GeneralAlarms.sErrorString:='Pozycja podnośnika dozowników jest poniżej ustawionej';	
END_IF
	
//Alarm_0044	44	Error	Stacja przeciągania dozowniki prawe | Pozycja podnośnika dozowników jest poniżej ustawionej
//BŁĄD 81 		
IF tonbFormsDragingRightRunCheck.Q THEN
	IF NOT arfbAlarm[44].bActive THEN
		arfbAlarm[44].Raise(nTimeStamp:=0);
	END_IF
	ELSE	
	IF arfbAlarm[44].bActive AND GeneralAlarms.bReset THEN
		arfbAlarm[44].Clear(nTimeStamp:=0, bResetConfirmation:= FALSE);	
	END_IF
// 	GeneralAlarms.bError:=TRUE;
// 	GeneralAlarms.bReset:=FALSE;
// 	GeneralAlarms.nErrorCode:=81;
// 	GeneralAlarms.sStationName:='Stacja przeciągania dozowniki prawe';
// 	GeneralAlarms.sErrorString:='Pozycja podnośnika dozowników jest poniżej ustawionej';	
END_IF

//Alarm_0045	45	Error	Brak kapsla/lub kilku pod rząd przed stacją ROPP , nałóż kapsle na butelki
//BŁĄD 368 - Brak nasadek po sorterze 
IF (iROPPFeederCheckCountNOK >= 1 AND bROPPCappingEnable ) THEN
	IF NOT arfbAlarm[45].bActive THEN
		arfbAlarm[45].Raise(nTimeStamp:=0);
	END_IF
	ELSE	
	IF arfbAlarm[45].bActive AND GeneralAlarms.bReset THEN
		arfbAlarm[45].Clear(nTimeStamp:=0, bResetConfirmation:= FALSE);	
	END_IF
// 	GeneralAlarms.bError:=TRUE;
// 	GeneralAlarms.bReset:=FALSE;
// 	GeneralAlarms.nErrorCode:=368;
// 	GeneralAlarms.udiStationID:=1;	
// 	GeneralAlarms.sStationName:='Błąd systemu';
// 	GeneralAlarms.sErrorString:='Brak kapsla/lub kilku pod rząd przed stacją ROPP ';
END_IF

//Alarm_0046	46	Error	Stacja ROPP | Zablokowana formatka za ROPP
//BŁĄD 369 -	Zablokowana formatka za stacją ROPP
IF (tonFormsStuckAfterROPPAlarm.Q) THEN
	IF NOT arfbAlarm[46].bActive THEN
		arfbAlarm[46].Raise(nTimeStamp:=0);
	END_IF
	ELSE	
	IF arfbAlarm[46].bActive AND GeneralAlarms.bReset THEN
		arfbAlarm[46].Clear(nTimeStamp:=0, bResetConfirmation:= FALSE);	
	END_IF
// 	GeneralAlarms.bError:=TRUE;
// 	GeneralAlarms.bReset:=FALSE;
// 	GeneralAlarms.nErrorCode:=369;
// 	GeneralAlarms.udiStationID:=1;	
// 	GeneralAlarms.sStationName:='Błąd systemu';
// 	GeneralAlarms.sErrorString:='Stacja ROPP | Zablokowana formatka za ROPP';
// 	GeneralAlarms.sErrorString2:='Stacja ROPP | Zablokowana formatka za ROPP';	
END_IF

//Alarm_0047	47	Error	Stacja zgrzewania platynek (opcja)| Zablokowana formatka za stacją		
//BŁĄD 370 -	Zablokowana formatka za stacją ROPP
IF (tonFormsStuckAfterLidSealerAlarm.Q) THEN
	IF NOT arfbAlarm[47].bActive THEN
		arfbAlarm[47].Raise(nTimeStamp:=0);
	END_IF
	ELSE	
	IF arfbAlarm[47].bActive AND GeneralAlarms.bReset THEN
		arfbAlarm[47].Clear(nTimeStamp:=0, bResetConfirmation:= FALSE);	
	END_IF
// 	GeneralAlarms.bError:=TRUE;
// 	GeneralAlarms.bReset:=FALSE;
// 	GeneralAlarms.nErrorCode:=370;
// 	GeneralAlarms.udiStationID:=1;	
// 	GeneralAlarms.sStationName:='Błąd systemu';
// 	GeneralAlarms.sErrorString:='Stacja zgrzewania platynek (opcja)| Zablokowana formatka za stacją';
// 	GeneralAlarms.sErrorString2:='Stacja zgrzewania platynek (opcja)| Zablokowana formatka za stacją';	
END_IF

//Alarm_0048	48	Error	Stacja sortera nakrętek | Zablokowana formatka za sorterem	
//BŁĄD 371 -	Zablokowana formatka przy stacji zakręcarek
IF (tonFormsStuckAfterCapSorterAlarm.Q) THEN
	IF NOT arfbAlarm[48].bActive THEN
		arfbAlarm[48].Raise(nTimeStamp:=0);
	END_IF
	ELSE	
	IF arfbAlarm[48].bActive AND GeneralAlarms.bReset THEN
		arfbAlarm[48].Clear(nTimeStamp:=0, bResetConfirmation:= FALSE);	
	END_IF
// 	GeneralAlarms.bError:=TRUE;
// 	GeneralAlarms.bReset:=FALSE;
// 	GeneralAlarms.nErrorCode:=371;
// 	GeneralAlarms.udiStationID:=1;	
// 	GeneralAlarms.sStationName:='Błąd systemu';
// 	GeneralAlarms.sErrorString:='Stacja sortera nakrętek | Zablokowana formatka za sorterem';
// 	GeneralAlarms.sErrorString2:='Stacja sortera nakrętek | Zablokowana formatka za sorterem';
END_IF

// Alarm_0049	49	Error	Stacja przeciągania dozowniki lewe | Formatki nie przeciągnięte	General
//BŁĄD  	
IF NOT VIS.bDosingTwoPhasesShow AND NOT bPhaseChanging AND (( P00_PackML.ftbFormsDragingLeftRun.Q AND NOT bDispencer12AllowDosingAfterDrag) 
	OR ( P00_PackML.ftbFormsDragingRightRun.Q AND NOT bDispencer34AllowDosingAfterDrag) 		)THEN
	IF NOT arfbAlarm[49].bActive THEN
		arfbAlarm[49].Raise(nTimeStamp:=0);
	END_IF
	ELSE	
	IF arfbAlarm[49].bActive AND GeneralAlarms.bReset THEN
		arfbAlarm[49].Clear(nTimeStamp:=0, bResetConfirmation:= FALSE);	
	END_IF
END_IF

// Alarm_0050	50	Error	Stacja przeciągania dozowniki prawe | Formatki nie przeciągnięte	General
//BŁĄD  	
//IF NOT VIS.bDosingTwoPhasesShow AND NOT bPhaseChanging AND(P00_PackML.ftbFormsDragingRightRun.Q AND NOT bDispencer34AllowDosingAfterDrag) THEN
//	IF NOT arfbAlarm[50].bActive THEN
//		arfbAlarm[50].Raise(nTimeStamp:=0);
//	END_IF
//	ELSE	
//	IF arfbAlarm[50].bActive AND GeneralAlarms.bReset THEN
//		arfbAlarm[50].Clear(nTimeStamp:=0, bResetConfirmation:= FALSE);	
//	END_IF
//END_IF

(*Wyświetlanie błedu na wyjściu*)
GeneralAlarms.bError				:= FALSE;
FOR nAlarmNumerator := 0 TO 79 DO
	GeneralAlarms.bError			:= GeneralAlarms.bError OR arfbAlarm[nAlarmNumerator].bActive;
END_FOR


//===================================================================================================


IF rtEmergencyStop.Q THEN
		bAllStationDoneDelay:=TRUE; 
END_IF
END_ACTION

ACTION aWarnings:
(**************** Warningi **************)
(************ Sygnały dla HMI ***********)

